  MoveL 728 to (114.51, 182.41, 0) mm, rotated rx 180 ry 0 rz -39.83 deg; joints [46.226, -66.396, 72.244, -0.865, 84.126, 46.311]
  MoveL 729 to (113.63, 182.75, 0) mm, rotated rx 180 ry 0 rz -39.83 deg; joints [46.185, -66.362, 72.194, -0.865, 84.141, 46.27]
  MoveL 730 to (112.75, 183.07, 0) mm, rotated rx 180 ry 0 rz -39.83 deg; joints [46.144, -66.329, 72.147, -0.865, 84.155, 46.229]
  MoveL 731 to (111.7, 183.43, 0) mm, rotated rx -180 ry 0 rz -39.83 deg; joints [46.095, -66.292, 72.093, -0.865, 84.171, 46.18]
  MoveL 732 to (110.64, 183.76, 0) mm, rotated rx 180 ry 0 rz -39.83 deg; joints [46.046, -66.257, 72.043, -0.865, 84.186, 46.13]
  MoveL 733 to (109.56, 184.05, 0) mm, rotated rx 180 ry 0 rz -39.83 deg; joints [45.995, -66.226, 71.997, -0.865, 84.199, 46.079]
  MoveL 734 to (108.47, 184.29, 0) mm, rotated rx 180 ry 0 rz -39.83 deg; joints [45.944, -66.198, 71.957, -0.864, 84.211, 46.028]
  MoveL 735 to (107.39, 184.47, 0) mm, rotated rx 180 ry 0 rz -39.83 deg; joints [45.893, -66.176, 71.924, -0.864, 84.221, 45.977]
  MoveL 736 to (106.3, 184.61, 0) mm, rotated rx 180 ry 0 rz -39.83 deg; joints [45.842, -66.158, 71.897, -0.864, 84.229, 45.925]
  MoveL 737 to (105.21, 184.7, 0) mm, rotated rx 180 ry 0 rz -39.83 deg; joints [45.79, -66.143, 71.874, -0.864, 84.236, 45.874]
  MoveL 738 to (104.14, 184.76, 0) mm, rotated rx 180 ry 0 rz -39.83 deg; joints [45.739, -66.13, 71.855, -0.864, 84.242, 45.822]
  MoveL 739 to (103.53, 184.79, 0) mm, rotated rx 180 ry 0 rz -39.83 deg; joints [45.71, -66.124, 71.846, -0.864, 84.245, 45.794]
  MoveL 740 to (102.92, 184.8, 0) mm, rotated rx 180 ry 0 rz -39.83 deg; joints [45.682, -66.119, 71.838, -0.864, 84.247, 45.765]
  MoveL 741 to (102.31, 184.8, 0) mm, rotated rx -180 ry 0 rz -39.83 deg; joints [45.652, -66.115, 71.832, -0.864, 84.249, 45.736]
  MoveL 742 to (101.69, 184.78, 0) mm, rotated rx -180 ry 0 rz -39.83 deg; joints [45.623, -66.113, 71.828, -0.864, 84.251, 45.706]
  MoveL 743 to (101.69, 184.78, 0) mm, rotated rx -180 ry 0 rz -39.83 deg; joints [45.623, -66.113, 71.828, -0.864, 84.251, 45.706]
  MoveL 744 to (101.07, 184.8, 0) mm, rotated rx 180 ry 0 rz -39.83 deg; joints [45.593, -66.107, 71.818, -0.864, 84.254, 45.676]
  MoveL 745 to (100.46, 184.8, 0) mm, rotated rx 180 ry 0 rz -39.83 deg; joints [45.564, -66.103, 71.811, -0.864, 84.256, 45.647]
  MoveL 746 to (99.86, 184.79, 0) mm, rotated rx -180 ry 0 rz -39.83 deg; joints [45.535, -66.1, 71.807, -0.864, 84.257, 45.618]
  MoveL 747 to (99.25, 184.76, 0) mm, rotated rx 180 ry 0 rz -39.83 deg; joints [45.506, -66.098, 71.803, -0.864, 84.258, 45.589]
  MoveL 748 to (98.18, 184.7, 0) mm, rotated rx 180 ry 0 rz -39.83 deg; joints [45.455, -66.096, 71.799, -0.864, 84.26, 45.538]
  MoveL 749 to (97.09, 184.61, 0) mm, rotated rx 180 ry 0 rz -39.83 deg; joints [45.403, -66.096, 71.798, -0.864, 84.26, 45.486]
  MoveL 750 to (96, 184.47, 0) mm, rotated rx -180 ry 0 rz -39.83 deg; joints [45.35, -66.1, 71.802, -0.864, 84.259, 45.433]
  MoveL 751 to (94.92, 184.29, 0) mm, rotated rx -180 ry 0 rz -39.83 deg; joints [45.298, -66.108, 71.812, -0.864, 84.257, 45.381]
  MoveL 752 to (93.83, 184.05, 0) mm, rotated rx 180 ry 0 rz -39.83 deg; joints [45.245, -66.121, 71.829, -0.864, 84.252, 45.328]
  MoveL 753 to (92.75, 183.76, 0) mm, rotated rx -180 ry 0 rz -39.83 deg; joints [45.193, -66.138, 71.852, -0.864, 84.245, 45.276]
  MoveL 754 to (91.69, 183.43, 0) mm, rotated rx -180 ry 0 rz -39.83 deg; joints [45.141, -66.159, 71.879, -0.864, 84.237, 45.224]
  MoveL 755 to (90.64, 183.07, 0) mm, rotated rx 180 ry 0 rz -39.83 deg; joints [45.089, -66.182, 71.911, -0.864, 84.229, 45.172]
  MoveL 756 to (89.75, 182.75, 0) mm, rotated rx 180 ry 0 rz -39.83 deg; joints [45.046, -66.203, 71.939, -0.864, 84.22, 45.129]
  MoveL 757 to (88.88, 182.41, 0) mm, rotated rx 180 ry 0 rz -39.83 deg; joints [45.003, -66.226, 71.97, -0.864, 84.211, 45.086]
  MoveL 758 to (88.02, 182.04, 0) mm, rotated rx -180 ry 0 rz -39.83 deg; joints [44.96, -66.251, 72.004, -0.864, 84.202, 45.044]
  MoveL 759 to (87.16, 181.64, 0) mm, rotated rx 180 ry 0 rz -39.83 deg; joints [44.917, -66.278, 72.042, -0.864, 84.191, 45.001]
  MoveL 760 to (86.31, 181.19, 0) mm, rotated rx 180 ry 0 rz -39.83 deg; joints [44.875, -66.31, 72.086, -0.864, 84.178, 44.959]
  MoveL 761 to (85.46, 180.71, 0) mm, rotated rx 180 ry 0 rz -39.83 deg; joints [44.832, -66.345, 72.134, -0.864, 84.164, 44.916]
  MoveL 762 to (84.63, 180.2, 0) mm, rotated rx 180 ry 0 rz -39.83 deg; joints [44.79, -66.382, 72.185, -0.864, 84.149, 44.875]
  MoveL 763 to (83.81, 179.68, 0) mm, rotated rx 180 ry 0 rz -39.83 deg; joints [44.749, -66.421, 72.239, -0.864, 84.134, 44.833]
  MoveL 764 to (83.1, 179.21, 0) mm, rotated rx 180 ry 0 rz -39.83 deg; joints [44.713, -66.455, 72.287, -0.864, 84.12, 44.798]
  MoveL 765 to (82.4, 178.72, 0) mm, rotated rx -180 ry 0 rz -39.83 deg; joints [44.677, -66.491, 72.336, -0.864, 84.106, 44.762]
  MoveL 766 to (81.72, 178.23, 0) mm, rotated rx 180 ry 0 rz -39.83 deg; joints [44.642, -66.528, 72.388, -0.864, 84.091, 44.727]
  MoveL 767 to (81.05, 177.71, 0) mm, rotated rx -180 ry 0 rz -39.83 deg; joints [44.608, -66.567, 72.441, -0.864, 84.076, 44.693]
  MoveL 768 to (80.23, 177.02, 0) mm, rotated rx 180 ry 0 rz -39.83 deg; joints [44.566, -66.619, 72.514, -0.864, 84.055, 44.651]
  MoveL 769 to (79.45, 176.29, 0) mm, rotated rx 180 ry 0 rz -39.83 deg; joints [44.525, -66.675, 72.591, -0.864, 84.033, 44.611]
  MoveL 770 to (78.71, 175.53, 0) mm, rotated rx -180 ry 0 rz -39.83 deg; joints [44.486, -66.734, 72.673, -0.864, 84.009, 44.572]
  MoveL 771 to (78.02, 174.73, 0) mm, rotated rx 180 ry 0 rz -39.83 deg; joints [44.449, -66.797, 72.76, -0.864, 83.984, 44.536]
  MoveL 772 to (77.69, 174.31, 0) mm, rotated rx 180 ry 0 rz -39.83 deg; joints [44.431, -66.83, 72.806, -0.864, 83.971, 44.518]
  MoveL 773 to (77.38, 173.88, 0) mm, rotated rx -180 ry 0 rz -39.83 deg; joints [44.414, -66.864, 72.854, -0.864, 83.957, 44.501]
  MoveL 774 to (77.09, 173.42, 0) mm, rotated rx 180 ry 0 rz -39.83 deg; joints [44.398, -66.901, 72.905, -0.864, 83.943, 44.485]
  MoveL 775 to (76.83, 172.93, 0) mm, rotated rx -180 ry 0 rz -39.83 deg; joints [44.383, -66.94, 72.96, -0.864, 83.927, 44.471]
  MoveL 776 to (76.65, 172.52, 0) mm, rotated rx 180 ry 0 rz -39.83 deg; joints [44.373, -66.974, 73.007, -0.864, 83.913, 44.46]
  MoveL 777 to (76.49, 172.09, 0) mm, rotated rx -180 ry 0 rz -39.83 deg; joints [44.363, -67.009, 73.056, -0.864, 83.899, 44.451]
  MoveL 778 to (76.36, 171.66, 0) mm, rotated rx 180 ry 0 rz -39.83 deg; joints [44.355, -67.045, 73.106, -0.864, 83.885, 44.443]
  MoveL 779 to (76.26, 171.24, 0) mm, rotated rx -180 ry 0 rz -39.83 deg; joints [44.348, -67.08, 73.155, -0.864, 83.871, 44.436]
  MoveL 780 to (76.2, 170.92, 0) mm, rotated rx 180 ry 0 rz -39.83 deg; joints [44.343, -67.107, 73.192, -0.864, 83.861, 44.432]
  MoveL 781 to (76.15, 170.61, 0) mm, rotated rx -180 ry 0 rz -39.83 deg; joints [44.339, -67.133, 73.229, -0.864, 83.85, 44.428]
  MoveL 782 to (76.11, 170.29, 0) mm, rotated rx 180 ry 0 rz -39.83 deg; joints [44.336, -67.16, 73.266, -0.864, 83.84, 44.425]
  MoveL 783 to (76.08, 169.97, 0) mm, rotated rx 180 ry 0 rz -39.83 deg; joints [44.333, -67.187, 73.304, -0.864, 83.829, 44.422]
  MoveL 784 to (76.06, 169.58, 0) mm, rotated rx 180 ry 0 rz -39.83 deg; joints [44.33, -67.22, 73.35, -0.864, 83.816, 44.419]
  MoveL 785 to (76.05, 169.18, 0) mm, rotated rx 180 ry 0 rz -39.83 deg; joints [44.327, -67.254, 73.397, -0.864, 83.802, 44.417]
  MoveL 786 to (76.05, 168.78, 0) mm, rotated rx 180 ry 0 rz -39.83 deg; joints [44.325, -67.288, 73.445, -0.864, 83.788, 44.415]
  MoveL 787 to (76.07, 168.37, 0) mm, rotated rx 180 ry 0 rz -39.83 deg; joints [44.324, -67.323, 73.494, -0.864, 83.775, 44.414]
  MoveL 788 to (76.11, 167.98, 0) mm, rotated rx -180 ry 0 rz -39.83 deg; joints [44.324, -67.356, 73.541, -0.864, 83.761, 44.415]
  MoveL 789 to (76.17, 167.59, 0) mm, rotated rx 180 ry 0 rz -39.83 deg; joints [44.325, -67.39, 73.588, -0.864, 83.748, 44.416]
  MoveL 790 to (76.26, 167.21, 0) mm, rotated rx -180 ry 0 rz -39.83 deg; joints [44.328, -67.423, 73.634, -0.864, 83.735, 44.418]
  MoveL 791 to (76.37, 166.84, 0) mm, rotated rx 180 ry 0 rz -39.83 deg; joints [44.331, -67.456, 73.679, -0.864, 83.722, 44.422]
  MoveL 792 to (76.54, 166.39, 0) mm, rotated rx -180 ry 0 rz -39.83 deg; joints [44.337, -67.495, 73.734, -0.864, 83.707, 44.428]
  MoveL 793 to (76.74, 165.96, 0) mm, rotated rx -180 ry 0 rz -39.83 deg; joints [44.345, -67.534, 73.789, -0.864, 83.691, 44.436]
  MoveL 794 to (76.97, 165.53, 0) mm, rotated rx -180 ry 0 rz -39.83 deg; joints [44.354, -67.572, 73.842, -0.864, 83.676, 44.445]
  MoveL 795 to (77.22, 165.11, 0) mm, rotated rx 180 ry 0 rz -39.83 deg; joints [44.364, -67.61, 73.895, -0.864, 83.661, 44.456]
  MoveL 796 to (77.53, 164.64, 0) mm, rotated rx -180 ry 0 rz -39.83 deg; joints [44.376, -67.653, 73.955, -0.864, 83.644, 44.468]
  MoveL 797 to (77.86, 164.18, 0) mm, rotated rx 180 ry 0 rz -39.83 deg; joints [44.39, -67.694, 74.014, -0.864, 83.628, 44.482]
  MoveL 798 to (78.2, 163.73, 0) mm, rotated rx -180 ry 0 rz -39.83 deg; joints [44.404, -67.735, 74.071, -0.864, 83.612, 44.497]
  MoveL 799 to (78.57, 163.3, 0) mm, rotated rx 180 ry 0 rz -39.83 deg; joints [44.42, -67.774, 74.126, -0.864, 83.596, 44.513]
  MoveL 800 to (79, 162.85, 0) mm, rotated rx -180 ry 0 rz -39.83 deg; joints [44.439, -67.817, 74.185, -0.864, 83.579, 44.532]
  MoveL 801 to (79.47, 162.42, 0) mm, rotated rx 180 ry 0 rz -39.83 deg; joints [44.459, -67.857, 74.241, -0.864, 83.563, 44.552]
  MoveL 802 to (79.95, 162.01, 0) mm, rotated rx 180 ry 0 rz -39.83 deg; joints [44.48, -67.896, 74.296, -0.865, 83.548, 44.574]
  MoveL 803 to (80.45, 161.62, 0) mm, rotated rx 180 ry 0 rz -39.83 deg; joints [44.503, -67.933, 74.348, -0.865, 83.534, 44.596]
  MoveL 804 to (81.09, 161.15, 0) mm, rotated rx 180 ry 0 rz -39.83 deg; joints [44.532, -67.978, 74.411, -0.865, 83.516, 44.626]
  MoveL 805 to (81.75, 160.71, 0) mm, rotated rx 180 ry 0 rz -39.83 deg; joints [44.562, -68.02, 74.471, -0.865, 83.499, 44.656]
  MoveL 806 to (82.43, 160.29, 0) mm, rotated rx 180 ry 0 rz -39.83 deg; joints [44.593, -68.061, 74.528, -0.865, 83.483, 44.687]
  MoveL 807 to (83.12, 159.89, 0) mm, rotated rx 180 ry 0 rz -39.83 deg; joints [44.624, -68.101, 74.584, -0.865, 83.467, 44.719]
  MoveL 808 to (83.7, 159.57, 0) mm, rotated rx 180 ry 0 rz -39.83 deg; joints [44.651, -68.133, 74.629, -0.865, 83.455, 44.746]
  MoveL 809 to (84.29, 159.25, 0) mm, rotated rx 180 ry 0 rz -39.83 deg; joints [44.678, -68.165, 74.673, -0.865, 83.442, 44.773]
  MoveL 810 to (84.89, 158.95, 0) mm, rotated rx 180 ry 0 rz -39.83 deg; joints [44.705, -68.195, 74.716, -0.865, 83.43, 44.801]
  MoveL 811 to (85.49, 158.67, 0) mm, rotated rx 180 ry 0 rz -39.83 deg; joints [44.734, -68.224, 74.757, -0.865, 83.419, 44.829]
  MoveL 812 to (86.31, 158.32, 0) mm, rotated rx 180 ry 0 rz -39.83 deg; joints [44.772, -68.26, 74.807, -0.865, 83.405, 44.868]
  MoveL 813 to (87.14, 157.99, 0) mm, rotated rx 180 ry 0 rz -39.83 deg; joints [44.811, -68.293, 74.855, -0.865, 83.392, 44.907]
  MoveL 814 to (87.99, 157.69, 0) mm, rotated rx 180 ry 0 rz -39.83 deg; joints [44.85, -68.325, 74.9, -0.865, 83.379, 44.946]
  MoveL 815 to (88.83, 157.41, 0) mm, rotated rx 180 ry 0 rz -39.83 deg; joints [44.89, -68.356, 74.943, -0.865, 83.367, 44.987]
  MoveL 816 to (89.62, 157.16, 0) mm, rotated rx -180 ry 0 rz -39.83 deg; joints [44.927, -68.383, 74.981, -0.865, 83.356, 45.024]
  MoveL 817 to (90.4, 156.92, 0) mm, rotated rx 180 ry 0 rz -39.83 deg; joints [44.964, -68.409, 75.018, -0.865, 83.346, 45.061]
  MoveL 818 to (91.19, 156.7, 0) mm, rotated rx 180 ry 0 rz -39.83 deg; joints [45.002, -68.434, 75.053, -0.865, 83.336, 45.099]
  MoveL 819 to (91.99, 156.5, 0) mm, rotated rx 180 ry 0 rz -39.83 deg; joints [45.04, -68.457, 75.086, -0.865, 83.327, 45.137]
  MoveL 820 to (92.82, 156.31, 0) mm, rotated rx 180 ry 0 rz -39.83 deg; joints [45.08, -68.479, 75.118, -0.865, 83.318, 45.177]
  MoveL 821 to (93.66, 156.14, 0) mm, rotated rx 180 ry 0 rz -39.83 deg; joints [45.12, -68.499, 75.147, -0.865, 83.31, 45.217]
  MoveL 822 to (94.51, 155.99, 0) mm, rotated rx 180 ry 0 rz -39.83 deg; joints [45.16, -68.518, 75.174, -0.865, 83.302, 45.258]
  MoveL 823 to (95.35, 155.86, 0) mm, rotated rx 180 ry 0 rz -39.83 deg; joints [45.201, -68.535, 75.199, -0.866, 83.295, 45.298]
  MoveL 824 to (96.38, 155.71, 0) mm, rotated rx 180 ry 0 rz -39.83 deg; joints [45.25, -68.555, 75.227, -0.866, 83.288, 45.348]
  MoveL 825 to (97.41, 155.59, 0) mm, rotated rx 180 ry 0 rz -39.83 deg; joints [45.3, -68.572, 75.252, -0.866, 83.28, 45.398]
  MoveL 826 to (98.44, 155.49, 0) mm, rotated rx -180 ry 0 rz -39.83 deg; joints [45.35, -68.588, 75.275, -0.866, 83.274, 45.448]
  MoveL 827 to (99.47, 155.42, 0) mm, rotated rx 180 ry 0 rz -39.83 deg; joints [45.4, -68.601, 75.294, -0.866, 83.269, 45.498]
  MoveL 828 to (100.02, 155.4, 0) mm, rotated rx 180 ry 0 rz -39.83 deg; joints [45.427, -68.606, 75.303, -0.866, 83.266, 45.525]
  MoveL 829 to (100.58, 155.38, 0) mm, rotated rx 180 ry 0 rz -39.83 deg; joints [45.454, -68.612, 75.311, -0.866, 83.264, 45.552]
  MoveL 830 to (101.14, 155.37, 0) mm, rotated rx -180 ry 0 rz -39.83 deg; joints [45.481, -68.616, 75.318, -0.866, 83.262, 45.579]
  MoveL 831 to (101.69, 155.36, 0) mm, rotated rx 180 ry 0 rz -39.83 deg; joints [45.508, -68.621, 75.325, -0.866, 83.26, 45.607]
  Establecer velocidad (1000.0 mm/s)
  MoveL 832 to (101.69, 155.36, 0) mm, rotated rx 180 ry 0 rz -39.83 deg; joints [45.508, -68.621, 75.325, -0.866, 83.26, 45.607]
  MoveL 833 to (101.69, 155.36, 20) mm, rotated rx 180 ry 0 rz -39.83 deg; joints [45.523, -68.888, 73.963, -0.863, 84.889, 45.597]

--- program P_in_2 (robot KUKA KR 16 2) ---
  Suave(1)
  Establecer velocidad (1000.0 mm/s)
  Est. Ref.: Frame 2
  Est. herr: Plumon_ensamble
  Mostrar Plumon_ensamble
  MoveJ 1 to (138.11, 152.35, 20) mm, rotated rx -180 ry 0 rz -39.83 deg; joints [47.298, -69.343, 74.631, -0.864, 84.703, 47.375]
  MoveL 2 to (138.11, 152.35, 20) mm, rotated rx -180 ry 0 rz -39.83 deg; joints [47.298, -69.343, 74.631, -0.864, 84.703, 47.375]
  MoveL 3 to (138.11, 152.35, 0) mm, rotated rx 180 ry 0 rz -39.83 deg; joints [47.283, -69.071, 75.989, -0.867, 83.072, 47.385]
  MoveL 4 to (138.11, 152.35, 0) mm, rotated rx 180 ry 0 rz -39.83 deg; joints [47.283, -69.071, 75.989, -0.867, 83.072, 47.385]
  Establecer velocidad (50.0 mm/s)
  MoveL 5 to (138.89, 152.07, 0) mm, rotated rx -180 ry 0 rz -39.83 deg; joints [47.321, -69.098, 76.027, -0.867, 83.062, 47.422]
  MoveL 6 to (139.65, 151.76, 0) mm, rotated rx -180 ry 0 rz -39.83 deg; joints [47.358, -69.127, 76.067, -0.867, 83.051, 47.459]
  MoveL 7 to (140.41, 151.43, 0) mm, rotated rx 180 ry 0 rz -39.83 deg; joints [47.394, -69.157, 76.11, -0.867, 83.039, 47.496]
  MoveL 8 to (141.16, 151.09, 0) mm, rotated rx 180 ry 0 rz -39.83 deg; joints [47.43, -69.189, 76.155, -0.867, 83.027, 47.532]
  MoveL 9 to (142.11, 150.62, 0) mm, rotated rx 180 ry 0 rz -39.83 deg; joints [47.476, -69.232, 76.215, -0.867, 83.011, 47.578]
  MoveL 10 to (143.04, 150.14, 0) mm, rotated rx 180 ry 0 rz -39.83 deg; joints [47.521, -69.277, 76.276, -0.867, 82.994, 47.623]
  MoveL 11 to (143.96, 149.63, 0) mm, rotated rx -180 ry 0 rz -39.83 deg; joints [47.565, -69.323, 76.341, -0.867, 82.977, 47.668]
  MoveL 12 to (144.87, 149.1, 0) mm, rotated rx 180 ry 0 rz -39.83 deg; joints [47.609, -69.37, 76.407, -0.867, 82.959, 47.712]
  MoveL 13 to (146, 148.42, 0) mm, rotated rx 180 ry 0 rz -39.83 deg; joints [47.663, -69.432, 76.492, -0.867, 82.936, 47.766]
  MoveL 14 to (147.1, 147.68, 0) mm, rotated rx 180 ry 0 rz -39.83 deg; joints [47.716, -69.498, 76.583, -0.867, 82.912, 47.819]
  MoveL 15 to (148.15, 146.89, 0) mm, rotated rx 180 ry 0 rz -39.83 deg; joints [47.766, -69.568, 76.68, -0.867, 82.886, 47.87]
  MoveL 16 to (149.12, 146.01, 0) mm, rotated rx 180 ry 0 rz -39.83 deg; joints [47.812, -69.645, 76.786, -0.867, 82.858, 47.916]
  MoveL 17 to (149.82, 145.25, 0) mm, rotated rx 180 ry 0 rz -39.83 deg; joints [47.845, -69.712, 76.877, -0.867, 82.834, 47.95]
  MoveL 18 to (150.48, 144.46, 0) mm, rotated rx 180 ry 0 rz -39.83 deg; joints [47.876, -69.781, 76.972, -0.867, 82.809, 47.982]
  MoveL 19 to (151.13, 143.64, 0) mm, rotated rx 180 ry 0 rz -39.83 deg; joints [47.907, -69.852, 77.069, -0.868, 82.783, 48.013]
  MoveL 20 to (151.78, 142.82, 0) mm, rotated rx -180 ry 0 rz -39.83 deg; joints [47.937, -69.923, 77.165, -0.868, 82.758, 48.043]
  MoveL 21 to (152.63, 141.8, 0) mm, rotated rx -180 ry 0 rz -39.83 deg; joints [47.978, -70.011, 77.286, -0.868, 82.726, 48.084]
  MoveL 22 to (153.49, 140.78, 0) mm, rotated rx -180 ry 0 rz -39.83 deg; joints [48.019, -70.099, 77.405, -0.868, 82.695, 48.126]
  MoveL 23 to (154.33, 139.76, 0) mm, rotated rx 180 ry 0 rz -39.83 deg; joints [48.058, -70.187, 77.526, -0.868, 82.663, 48.166]
  MoveL 24 to (155.11, 138.69, 0) mm, rotated rx 180 ry 0 rz -39.83 deg; joints [48.095, -70.279, 77.651, -0.868, 82.631, 48.203]
  MoveL 25 to (155.71, 137.74, 0) mm, rotated rx 180 ry 0 rz -39.83 deg; joints [48.123, -70.361, 77.761, -0.868, 82.602, 48.232]
  MoveL 26 to (156.26, 136.75, 0) mm, rotated rx 180 ry 0 rz -39.83 deg; joints [48.149, -70.445, 77.876, -0.868, 82.573, 48.258]
  MoveL 27 to (156.76, 135.74, 0) mm, rotated rx -180 ry 0 rz -39.83 deg; joints [48.172, -70.532, 77.993, -0.868, 82.543, 48.282]
  MoveL 28 to (157.24, 134.7, 0) mm, rotated rx 180 ry 0 rz -39.83 deg; joints [48.194, -70.62, 78.111, -0.868, 82.512, 48.304]
  MoveL 29 to (157.83, 133.33, 0) mm, rotated rx -180 ry 0 rz -39.83 deg; joints [48.222, -70.736, 78.268, -0.868, 82.472, 48.332]
  MoveL 30 to (158.37, 131.95, 0) mm, rotated rx 180 ry 0 rz -39.83 deg; joints [48.246, -70.853, 78.426, -0.868, 82.432, 48.358]
  MoveL 31 to (158.85, 130.54, 0) mm, rotated rx 180 ry 0 rz -39.83 deg; joints [48.268, -70.972, 78.586, -0.868, 82.392, 48.38]
  MoveL 32 to (159.24, 129.11, 0) mm, rotated rx 180 ry 0 rz -39.83 deg; joints [48.285, -71.093, 78.747, -0.868, 82.351, 48.397]
  MoveL 33 to (159.49, 127.9, 0) mm, rotated rx 180 ry 0 rz -39.83 deg; joints [48.296, -71.195, 78.883, -0.868, 82.317, 48.408]
  MoveL 34 to (159.67, 126.67, 0) mm, rotated rx 180 ry 0 rz -39.83 deg; joints [48.303, -71.298, 79.021, -0.868, 82.283, 48.416]
  MoveL 35 to (159.81, 125.43, 0) mm, rotated rx 180 ry 0 rz -39.83 deg; joints [48.308, -71.402, 79.159, -0.869, 82.249, 48.422]
  MoveL 36 to (159.9, 124.19, 0) mm, rotated rx -180 ry 0 rz -39.83 deg; joints [48.31, -71.506, 79.297, -0.869, 82.215, 48.425]
  MoveL 37 to (159.96, 123.02, 0) mm, rotated rx -180 ry 0 rz -39.83 deg; joints [48.311, -71.603, 79.426, -0.869, 82.183, 48.426]
  MoveL 38 to (159.99, 121.86, 0) mm, rotated rx 180 ry 0 rz -39.83 deg; joints [48.311, -71.701, 79.555, -0.869, 82.151, 48.426]
  MoveL 39 to (159.97, 120.69, 0) mm, rotated rx 180 ry 0 rz -39.83 deg; joints [48.308, -71.798, 79.684, -0.869, 82.12, 48.424]
  MoveL 40 to (159.9, 119.53, 0) mm, rotated rx 180 ry 0 rz -39.83 deg; joints [48.303, -71.894, 79.811, -0.869, 82.089, 48.419]
  MoveL 41 to (159.71, 117.85, 0) mm, rotated rx -180 ry 0 rz -39.83 deg; joints [48.29, -72.034, 79.995, -0.869, 82.044, 48.407]
  MoveL 42 to (159.41, 116.18, 0) mm, rotated rx 180 ry 0 rz -39.83 deg; joints [48.272, -72.172, 80.177, -0.869, 82.001, 48.39]
  MoveL 43 to (159.03, 114.52, 0) mm, rotated rx 180 ry 0 rz -39.83 deg; joints [48.25, -72.309, 80.357, -0.869, 81.958, 48.368]
  MoveL 44 to (158.57, 112.88, 0) mm, rotated rx -180 ry 0 rz -39.83 deg; joints [48.224, -72.445, 80.534, -0.869, 81.916, 48.343]
  MoveL 45 to (158.12, 111.47, 0) mm, rotated rx 180 ry 0 rz -39.83 deg; joints [48.198, -72.561, 80.686, -0.869, 81.88, 48.318]
  MoveL 46 to (157.6, 110.08, 0) mm, rotated rx 180 ry 0 rz -39.83 deg; joints [48.169, -72.676, 80.835, -0.869, 81.845, 48.29]
  MoveL 47 to (157, 108.73, 0) mm, rotated rx -180 ry 0 rz -39.83 deg; joints [48.136, -72.786, 80.978, -0.869, 81.811, 48.257]
  MoveL 48 to (156.31, 107.43, 0) mm, rotated rx 180 ry 0 rz -39.83 deg; joints [48.098, -72.892, 81.116, -0.87, 81.779, 48.219]
  MoveL 49 to (155.34, 105.97, 0) mm, rotated rx -180 ry 0 rz -39.83 deg; joints [48.046, -73.01, 81.268, -0.87, 81.744, 48.168]
  MoveL 50 to (154.22, 104.62, 0) mm, rotated rx 180 ry 0 rz -39.83 deg; joints [47.986, -73.119, 81.408, -0.87, 81.712, 48.108]
  MoveL 51 to (152.99, 103.37, 0) mm, rotated rx 180 ry 0 rz -39.83 deg; joints [47.92, -73.219, 81.536, -0.87, 81.683, 48.043]
  MoveL 52 to (151.65, 102.24, 0) mm, rotated rx 180 ry 0 rz -39.83 deg; joints [47.849, -73.309, 81.651, -0.87, 81.657, 47.972]
  MoveL 53 to (150.39, 101.33, 0) mm, rotated rx 180 ry 0 rz -39.83 deg; joints [47.783, -73.38, 81.742, -0.87, 81.636, 47.906]
  MoveL 54 to (149.08, 100.52, 0) mm, rotated rx 180 ry 0 rz -39.83 deg; joints [47.713, -73.443, 81.821, -0.87, 81.619, 47.837]
  MoveL 55 to (147.72, 99.8, 0) mm, rotated rx -180 ry 0 rz -39.83 deg; joints [47.642, -73.498, 81.891, -0.87, 81.603, 47.765]
  MoveL 56 to (146.32, 99.18, 0) mm, rotated rx 180 ry 0 rz -39.83 deg; joints [47.568, -73.545, 81.95, -0.87, 81.59, 47.692]
  MoveL 57 to (145.08, 98.71, 0) mm, rotated rx 180 ry 0 rz -39.83 deg; joints [47.503, -73.579, 81.992, -0.87, 81.581, 47.627]
  MoveL 58 to (143.83, 98.32, 0) mm, rotated rx 180 ry 0 rz -39.83 deg; joints [47.437, -73.607, 82.027, -0.87, 81.573, 47.562]
  MoveL 59 to (142.55, 97.98, 0) mm, rotated rx 180 ry 0 rz -39.83 deg; joints [47.371, -73.63, 82.055, -0.87, 81.567, 47.495]
  MoveL 60 to (141.26, 97.71, 0) mm, rotated rx 180 ry 0 rz -39.83 deg; joints [47.303, -73.647, 82.075, -0.87, 81.563, 47.428]
  MoveL 61 to (139.77, 97.48, 0) mm, rotated rx -180 ry 0 rz -39.83 deg; joints [47.226, -73.661, 82.091, -0.87, 81.56, 47.35]
  MoveL 62 to (138.27, 97.33, 0) mm, rotated rx 180 ry 0 rz -39.83 deg; joints [47.148, -73.667, 82.097, -0.87, 81.559, 47.273]
  MoveL 63 to (136.77, 97.27, 0) mm, rotated rx 180 ry 0 rz -39.83 deg; joints [47.07, -73.666, 82.093, -0.87, 81.56, 47.195]
  MoveL 64 to (135.27, 97.31, 0) mm, rotated rx 180 ry 0 rz -39.83 deg; joints [46.993, -73.656, 82.078, -0.87, 81.564, 47.117]
  MoveL 65 to (133.81, 97.45, 0) mm, rotated rx 180 ry 0 rz -39.83 deg; joints [46.919, -73.638, 82.054, -0.87, 81.57, 47.043]
  MoveL 66 to (132.37, 97.68, 0) mm, rotated rx 180 ry 0 rz -39.83 deg; joints [46.845, -73.613, 82.019, -0.87, 81.578, 46.969]
  MoveL 67 to (130.95, 97.99, 0) mm, rotated rx 180 ry 0 rz -39.83 deg; joints [46.773, -73.58, 81.975, -0.87, 81.588, 46.896]
  MoveL 68 to (129.54, 98.38, 0) mm, rotated rx 180 ry 0 rz -39.83 deg; joints [46.701, -73.542, 81.923, -0.87, 81.6, 46.825]
  MoveL 69 to (128.37, 98.76, 0) mm, rotated rx 180 ry 0 rz -39.83 deg; joints [46.642, -73.504, 81.874, -0.87, 81.612, 46.766]
  MoveL 70 to (127.22, 99.19, 0) mm, rotated rx -180 ry 0 rz -39.83 deg; joints [46.584, -73.463, 81.818, -0.87, 81.624, 46.708]
  MoveL 71 to (126.1, 99.69, 0) mm, rotated rx 180 ry 0 rz -39.83 deg; joints [46.528, -73.416, 81.757, -0.87, 81.639, 46.651]
  MoveL 72 to (125.01, 100.24, 0) mm, rotated rx -180 ry 0 rz -39.83 deg; joints [46.474, -73.365, 81.689, -0.87, 81.654, 46.597]
  MoveL 73 to (123.6, 101.09, 0) mm, rotated rx 180 ry 0 rz -39.83 deg; joints [46.405, -73.288, 81.587, -0.869, 81.678, 46.527]
  MoveL 74 to (122.25, 102.03, 0) mm, rotated rx 180 ry 0 rz -39.83 deg; joints [46.339, -73.203, 81.475, -0.869, 81.704, 46.461]
  MoveL 75 to (120.95, 103.04, 0) mm, rotated rx 180 ry 0 rz -39.83 deg; joints [46.275, -73.112, 81.355, -0.869, 81.732, 46.397]
  MoveL 76 to (119.68, 104.1, 0) mm, rotated rx 180 ry 0 rz -39.83 deg; joints [46.214, -73.017, 81.23, -0.869, 81.761, 46.335]
  MoveL 77 to (118.34, 105.29, 0) mm, rotated rx -180 ry 0 rz -39.83 deg; joints [46.15, -72.911, 81.09, -0.869, 81.794, 46.27]
  MoveL 78 to (117.04, 106.52, 0) mm, rotated rx -180 ry 0 rz -39.83 deg; joints [46.088, -72.801, 80.946, -0.869, 81.828, 46.208]
  MoveL 79 to (115.79, 107.81, 0) mm, rotated rx 180 ry 0 rz -39.83 deg; joints [46.029, -72.688, 80.796, -0.869, 81.864, 46.148]
  MoveL 80 to (114.62, 109.16, 0) mm, rotated rx 180 ry 0 rz -39.83 deg; joints [45.974, -72.569, 80.639, -0.869, 81.901, 46.093]
  MoveL 81 to (113.74, 110.29, 0) mm, rotated rx 180 ry 0 rz -39.83 deg; joints [45.934, -72.469, 80.507, -0.869, 81.932, 46.052]
  MoveL 82 to (112.92, 111.47, 0) mm, rotated rx -180 ry 0 rz -39.83 deg; joints [45.896, -72.366, 80.371, -0.869, 81.965, 46.014]
  MoveL 83 to (112.15, 112.69, 0) mm, rotated rx 180 ry 0 rz -39.83 deg; joints [45.862, -72.26, 80.231, -0.869, 81.999, 45.979]
  MoveL 84 to (111.43, 113.95, 0) mm, rotated rx -180 ry 0 rz -39.83 deg; joints [45.83, -72.152, 80.088, -0.868, 82.033, 45.947]
  MoveL 85 to (110.6, 115.55, 0) mm, rotated rx 180 ry 0 rz -39.83 deg; joints [45.794, -72.013, 79.904, -0.868, 82.078, 45.911]
  MoveL 86 to (109.85, 117.2, 0) mm, rotated rx 180 ry 0 rz -39.83 deg; joints [45.763, -71.872, 79.716, -0.868, 82.123, 45.879]
  MoveL 87 to (109.19, 118.88, 0) mm, rotated rx 180 ry 0 rz -39.83 deg; joints [45.736, -71.728, 79.525, -0.868, 82.17, 45.851]
  MoveL 88 to (108.63, 120.6, 0) mm, rotated rx 180 ry 0 rz -39.83 deg; joints [45.715, -71.581, 79.33, -0.868, 82.218, 45.829]
  MoveL 89 to (108.12, 122.52, 0) mm, rotated rx 180 ry 0 rz -39.83 deg; joints [45.697, -71.418, 79.112, -0.868, 82.272, 45.81]
  MoveL 90 to (107.73, 124.48, 0) mm, rotated rx 180 ry 0 rz -39.83 deg; joints [45.685, -71.252, 78.892, -0.868, 82.327, 45.797]
  MoveL 91 to (107.46, 126.46, 0) mm, rotated rx -180 ry 0 rz -39.83 deg; joints [45.679, -71.086, 78.67, -0.868, 82.382, 45.79]
  MoveL 92 to (107.3, 128.45, 0) mm, rotated rx -180 ry 0 rz -39.83 deg; joints [45.679, -70.918, 78.446, -0.867, 82.439, 45.789]
  MoveL 93 to (107.26, 129.89, 0) mm, rotated rx 180 ry 0 rz -39.83 deg; joints [45.682, -70.798, 78.285, -0.867, 82.479, 45.792]
  MoveL 94 to (107.28, 131.32, 0) mm, rotated rx 180 ry 0 rz -39.83 deg; joints [45.689, -70.678, 78.125, -0.867, 82.52, 45.799]
  MoveL 95 to (107.38, 132.75, 0) mm, rotated rx 180 ry 0 rz -39.83 deg; joints [45.7, -70.559, 77.965, -0.867, 82.561, 45.809]
  MoveL 96 to (107.56, 134.17, 0) mm, rotated rx -180 ry 0 rz -39.83 deg; joints [45.714, -70.442, 77.807, -0.867, 82.601, 45.823]
  MoveL 97 to (107.88, 135.74, 0) mm, rotated rx 180 ry 0 rz -39.83 deg; joints [45.736, -70.312, 77.634, -0.867, 82.646, 45.844]
  MoveL 98 to (108.3, 137.28, 0) mm, rotated rx 180 ry 0 rz -39.83 deg; joints [45.763, -70.185, 77.464, -0.867, 82.689, 45.87]
  MoveL 99 to (108.82, 138.8, 0) mm, rotated rx 180 ry 0 rz -39.83 deg; joints [45.795, -70.061, 77.297, -0.867, 82.733, 45.901]
  MoveL 100 to (109.43, 140.29, 0) mm, rotated rx 180 ry 0 rz -39.83 deg; joints [45.83, -69.94, 77.134, -0.867, 82.775, 45.936]
  MoveL 101 to (110.26, 142.02, 0) mm, rotated rx 180 ry 0 rz -39.83 deg; joints [45.878, -69.8, 76.945, -0.867, 82.824, 45.983]
  MoveL 102 to (111.22, 143.67, 0) mm, rotated rx 180 ry 0 rz -39.83 deg; joints [45.932, -69.667, 76.766, -0.867, 82.871, 46.036]
  MoveL 103 to (112.32, 145.24, 0) mm, rotated rx -180 ry 0 rz -39.83 deg; joints [45.991, -69.542, 76.597, -0.867, 82.915, 46.095]
  MoveL 104 to (113.56, 146.68, 0) mm, rotated rx 180 ry 0 rz -39.83 deg; joints [46.058, -69.428, 76.444, -0.867, 82.956, 46.161]
  MoveL 105 to (114.42, 147.52, 0) mm, rotated rx 180 ry 0 rz -39.83 deg; joints [46.103, -69.362, 76.355, -0.867, 82.979, 46.206]
  MoveL 106 to (115.34, 148.31, 0) mm, rotated rx 180 ry 0 rz -39.83 deg; joints [46.151, -69.301, 76.273, -0.867, 83.001, 46.253]
  MoveL 107 to (116.29, 149.04, 0) mm, rotated rx 180 ry 0 rz -39.83 deg; joints [46.201, -69.244, 76.197, -0.867, 83.021, 46.303]
  MoveL 108 to (117.29, 149.74, 0) mm, rotated rx -180 ry 0 rz -39.83 deg; joints [46.252, -69.191, 76.126, -0.867, 83.04, 46.353]
  MoveL 109 to (118.22, 150.33, 0) mm, rotated rx 180 ry 0 rz -39.83 deg; joints [46.3, -69.146, 76.066, -0.867, 83.056, 46.401]
  MoveL 110 to (119.17, 150.89, 0) mm, rotated rx 180 ry 0 rz -39.83 deg; joints [46.348, -69.104, 76.01, -0.867, 83.071, 46.449]
  MoveL 111 to (120.15, 151.4, 0) mm, rotated rx -180 ry 0 rz -39.83 deg; joints [46.398, -69.066, 75.959, -0.867, 83.084, 46.499]
  MoveL 112 to (121.15, 151.87, 0) mm, rotated rx 180 ry 0 rz -39.83 deg; joints [46.449, -69.033, 75.915, -0.867, 83.096, 46.549]
  MoveL 113 to (122.06, 152.23, 0) mm, rotated rx 180 ry 0 rz -39.83 deg; joints [46.494, -69.006, 75.88, -0.867, 83.105, 46.595]
  MoveL 114 to (122.98, 152.55, 0) mm, rotated rx 180 ry 0 rz -39.83 deg; joints [46.541, -68.984, 75.851, -0.867, 83.113, 46.641]
  MoveL 115 to (123.92, 152.83, 0) mm, rotated rx 180 ry 0 rz -39.83 deg; joints [46.588, -68.965, 75.826, -0.867, 83.119, 46.688]
  MoveL 116 to (124.88, 153.06, 0) mm, rotated rx -180 ry 0 rz -39.83 deg; joints [46.635, -68.951, 75.807, -0.867, 83.124, 46.736]
  MoveL 117 to (125.65, 153.22, 0) mm, rotated rx -180 ry 0 rz -39.83 deg; joints [46.674, -68.941, 75.796, -0.867, 83.127, 46.774]
  MoveL 118 to (126.43, 153.34, 0) mm, rotated rx -180 ry 0 rz -39.83 deg; joints [46.713, -68.935, 75.787, -0.867, 83.129, 46.813]
  MoveL 119 to (127.22, 153.45, 0) mm, rotated rx -180 ry 0 rz -39.83 deg; joints [46.751, -68.93, 75.782, -0.867, 83.13, 46.852]
  MoveL 120 to (128, 153.53, 0) mm, rotated rx 180 ry 0 rz -39.83 deg; joints [46.79, -68.926, 75.778, -0.867, 83.131, 46.89]
  MoveL 121 to (128.52, 153.58, 0) mm, rotated rx 180 ry 0 rz -39.83 deg; joints [46.816, -68.925, 75.777, -0.867, 83.131, 46.916]
  MoveL 122 to (129.05, 153.62, 0) mm, rotated rx 180 ry 0 rz -39.83 deg; joints [46.841, -68.924, 75.776, -0.867, 83.131, 46.942]
  MoveL 123 to (129.57, 153.65, 0) mm, rotated rx 180 ry 0 rz -39.83 deg; joints [46.867, -68.924, 75.777, -0.867, 83.131, 46.967]
  MoveL 124 to (130.09, 153.67, 0) mm, rotated rx 180 ry 0 rz -39.83 deg; joints [46.893, -68.925, 75.779, -0.867, 83.131, 46.993]
  MoveL 125 to (130.82, 153.67, 0) mm, rotated rx -180 ry 0 rz -39.83 deg; joints [46.928, -68.928, 75.784, -0.867, 83.129, 47.029]
  MoveL 126 to (131.54, 153.65, 0) mm, rotated rx 180 ry 0 rz -39.83 deg; joints [46.964, -68.933, 75.792, -0.867, 83.127, 47.065]
  MoveL 127 to (132.27, 153.6, 0) mm, rotated rx 180 ry 0 rz -39.83 deg; joints [47, -68.94, 75.803, -0.867, 83.124, 47.1]
  MoveL 128 to (132.99, 153.52, 0) mm, rotated rx 180 ry 0 rz -39.83 deg; joints [47.035, -68.95, 75.817, -0.867, 83.12, 47.135]
  MoveL 129 to (133.82, 153.39, 0) mm, rotated rx -180 ry 0 rz -39.83 deg; joints [47.075, -68.965, 75.838, -0.867, 83.114, 47.176]
  MoveL 130 to (134.82, 153.18, 0) mm, rotated rx 180 ry 0 rz -39.83 deg; joints [47.124, -68.987, 75.87, -0.867, 83.105, 47.225]
  MoveL 131 to (136.19, 152.85, 0) mm, rotated rx -180 ry 0 rz -39.83 deg; joints [47.19, -69.021, 75.918, -0.867, 83.092, 47.291]
  MoveL 132 to (138.11, 152.35, 0) mm, rotated rx 180 ry 0 rz -39.83 deg; joints [47.283, -69.071, 75.989, -0.867, 83.072, 47.385]
  Establecer velocidad (1000.0 mm/s)
  MoveL 133 to (138.11, 152.35, 0) mm, rotated rx 180 ry 0 rz -39.83 deg; joints [47.283, -69.071, 75.989, -0.867, 83.072, 47.385]
  MoveL 134 to (138.11, 152.35, 20) mm, rotated rx -180 ry 0 rz -39.83 deg; joints [47.298, -69.343, 74.631, -0.864, 84.703, 47.375]
  Establecer velocidad (1000.0 mm/s)
  MoveL 135 to (65.28, 152.35, 20) mm, rotated rx 180 ry 0 rz -39.83 deg; joints [43.733, -68.85, 73.864, -0.862, 84.923, 43.806]
  MoveL 136 to (65.28, 152.35, 0) mm, rotated rx 180 ry 0 rz -39.83 deg; joints [43.719, -68.584, 75.226, -0.864, 83.294, 43.816]
  MoveL 137 to (65.28, 152.35, 0) mm, rotated rx 180 ry 0 rz -39.83 deg; joints [43.719, -68.584, 75.226, -0.864, 83.294, 43.816]
  Establecer velocidad (50.0 mm/s)
  MoveL 138 to (64.5, 152.07, 0) mm, rotated rx -180 ry 0 rz -39.83 deg; joints [43.679, -68.6, 75.248, -0.864, 83.289, 43.777]
  MoveL 139 to (63.73, 151.76, 0) mm, rotated rx 180 ry 0 rz -39.83 deg; joints [43.64, -68.619, 75.272, -0.864, 83.282, 43.738]
  MoveL 140 to (62.97, 151.43, 0) mm, rotated rx 180 ry 0 rz -39.83 deg; joints [43.601, -68.639, 75.3, -0.864, 83.275, 43.699]
  MoveL 141 to (62.23, 151.09, 0) mm, rotated rx -180 ry 0 rz -39.83 deg; joints [43.563, -68.661, 75.329, -0.864, 83.267, 43.661]
  MoveL 142 to (61.28, 150.62, 0) mm, rotated rx 180 ry 0 rz -39.83 deg; joints [43.514, -68.691, 75.369, -0.864, 83.256, 43.612]
  MoveL 143 to (60.35, 150.14, 0) mm, rotated rx 180 ry 0 rz -39.83 deg; joints [43.466, -68.723, 75.412, -0.864, 83.245, 43.564]
  MoveL 144 to (59.43, 149.63, 0) mm, rotated rx 180 ry 0 rz -39.83 deg; joints [43.418, -68.757, 75.457, -0.864, 83.233, 43.516]
  MoveL 145 to (58.51, 149.1, 0) mm, rotated rx 180 ry 0 rz -39.83 deg; joints [43.371, -68.792, 75.504, -0.864, 83.22, 43.469]
  MoveL 146 to (57.39, 148.42, 0) mm, rotated rx 180 ry 0 rz -39.83 deg; joints [43.312, -68.839, 75.566, -0.864, 83.203, 43.41]
  MoveL 147 to (56.29, 147.68, 0) mm, rotated rx 180 ry 0 rz -39.83 deg; joints [43.254, -68.89, 75.634, -0.864, 83.185, 43.353]
  MoveL 148 to (55.24, 146.89, 0) mm, rotated rx 180 ry 0 rz -39.83 deg; joints [43.198, -68.946, 75.71, -0.864, 83.165, 43.297]
  MoveL 149 to (54.27, 146.01, 0) mm, rotated rx 180 ry 0 rz -39.83 deg; joints [43.146, -69.01, 75.797, -0.864, 83.142, 43.245]
  MoveL 150 to (53.57, 145.25, 0) mm, rotated rx -180 ry 0 rz -39.83 deg; joints [43.107, -69.067, 75.873, -0.864, 83.121, 43.206]
  MoveL 151 to (52.9, 144.46, 0) mm, rotated rx 180 ry 0 rz -39.83 deg; joints [43.069, -69.127, 75.954, -0.864, 83.1, 43.169]
  MoveL 152 to (52.26, 143.64, 0) mm, rotated rx 180 ry 0 rz -39.83 deg; joints [43.033, -69.189, 76.038, -0.864, 83.077, 43.133]
  MoveL 153 to (51.61, 142.82, 0) mm, rotated rx -180 ry 0 rz -39.83 deg; joints [42.996, -69.251, 76.122, -0.864, 83.055, 43.097]
  MoveL 154 to (50.76, 141.8, 0) mm, rotated rx 180 ry 0 rz -39.83 deg; joints [42.948, -69.328, 76.226, -0.864, 83.027, 43.049]
  MoveL 155 to (49.9, 140.78, 0) mm, rotated rx 180 ry 0 rz -39.83 deg; joints [42.899, -69.404, 76.328, -0.864, 83, 43.001]
  MoveL 156 to (49.06, 139.76, 0) mm, rotated rx 180 ry 0 rz -39.83 deg; joints [42.852, -69.481, 76.432, -0.864, 82.973, 42.954]
  MoveL 157 to (48.28, 138.69, 0) mm, rotated rx -180 ry 0 rz -39.83 deg; joints [42.807, -69.562, 76.541, -0.864, 82.944, 42.909]
  MoveL 158 to (47.68, 137.74, 0) mm, rotated rx 180 ry 0 rz -39.83 deg; joints [42.772, -69.635, 76.64, -0.864, 82.918, 42.874]
  MoveL 159 to (47.13, 136.75, 0) mm, rotated rx 180 ry 0 rz -39.83 deg; joints [42.738, -69.712, 76.743, -0.864, 82.891, 42.841]
  MoveL 160 to (46.63, 135.74, 0) mm, rotated rx 180 ry 0 rz -39.83 deg; joints [42.707, -69.791, 76.85, -0.864, 82.863, 42.81]
  MoveL 161 to (46.15, 134.7, 0) mm, rotated rx 180 ry 0 rz -39.83 deg; joints [42.677, -69.873, 76.96, -0.864, 82.834, 42.781]
  MoveL 162 to (45.56, 133.33, 0) mm, rotated rx 180 ry 0 rz -39.83 deg; joints [42.639, -69.981, 77.105, -0.864, 82.796, 42.743]
  MoveL 163 to (45.02, 131.95, 0) mm, rotated rx 180 ry 0 rz -39.83 deg; joints [42.603, -70.09, 77.252, -0.864, 82.758, 42.708]
  MoveL 164 to (44.54, 130.54, 0) mm, rotated rx 180 ry 0 rz -39.83 deg; joints [42.57, -70.202, 77.403, -0.864, 82.719, 42.676]
  MoveL 165 to (44.15, 129.11, 0) mm, rotated rx 180 ry 0 rz -39.83 deg; joints [42.542, -70.317, 77.557, -0.864, 82.679, 42.648]
  MoveL 166 to (43.9, 127.9, 0) mm, rotated rx -180 ry 0 rz -39.83 deg; joints [42.521, -70.416, 77.689, -0.864, 82.645, 42.628]
  MoveL 167 to (43.72, 126.67, 0) mm, rotated rx 180 ry 0 rz -39.83 deg; joints [42.504, -70.516, 77.824, -0.864, 82.611, 42.611]
  MoveL 168 to (43.58, 125.43, 0) mm, rotated rx 180 ry 0 rz -39.83 deg; joints [42.489, -70.617, 77.96, -0.864, 82.576, 42.597]
  MoveL 169 to (43.49, 124.19, 0) mm, rotated rx 180 ry 0 rz -39.83 deg; joints [42.476, -70.72, 78.097, -0.864, 82.541, 42.584]
  MoveL 170 to (43.43, 123.02, 0) mm, rotated rx -180 ry 0 rz -39.83 deg; joints [42.465, -70.816, 78.226, -0.864, 82.508, 42.574]
  MoveL 171 to (43.4, 121.86, 0) mm, rotated rx 180 ry 0 rz -39.83 deg; joints [42.456, -70.913, 78.355, -0.864, 82.476, 42.566]
  MoveL 172 to (43.42, 120.69, 0) mm, rotated rx 180 ry 0 rz -39.83 deg; joints [42.449, -71.009, 78.484, -0.864, 82.443, 42.559]
  MoveL 173 to (43.49, 119.53, 0) mm, rotated rx 180 ry 0 rz -39.83 deg; joints [42.445, -71.106, 78.614, -0.864, 82.411, 42.555]
  MoveL 174 to (43.68, 117.85, 0) mm, rotated rx 180 ry 0 rz -39.83 deg; joints [42.443, -71.248, 78.803, -0.864, 82.363, 42.554]
  MoveL 175 to (43.97, 116.18, 0) mm, rotated rx 180 ry 0 rz -39.83 deg; joints [42.446, -71.39, 78.992, -0.864, 82.316, 42.558]
  MoveL 176 to (44.36, 114.52, 0) mm, rotated rx 180 ry 0 rz -39.83 deg; joints [42.454, -71.531, 79.18, -0.864, 82.27, 42.567]
  MoveL 177 to (44.82, 112.88, 0) mm, rotated rx -180 ry 0 rz -39.83 deg; joints [42.466, -71.673, 79.368, -0.865, 82.223, 42.579]
  MoveL 178 to (45.27, 111.47, 0) mm, rotated rx 180 ry 0 rz -39.83 deg; joints [42.479, -71.795, 79.53, -0.865, 82.183, 42.593]
  MoveL 179 to (45.79, 110.08, 0) mm, rotated rx 180 ry 0 rz -39.83 deg; joints [42.496, -71.915, 79.69, -0.865, 82.144, 42.61]
  MoveL 180 to (46.38, 108.73, 0) mm, rotated rx 180 ry 0 rz -39.83 deg; joints [42.517, -72.034, 79.846, -0.865, 82.106, 42.632]
  MoveL 181 to (47.08, 107.43, 0) mm, rotated rx 180 ry 0 rz -39.83 deg; joints [42.543, -72.149, 79.999, -0.865, 82.069, 42.658]
  MoveL 182 to (48.05, 105.97, 0) mm, rotated rx 180 ry 0 rz -39.83 deg; joints [42.582, -72.279, 80.171, -0.865, 82.028, 42.698]
  MoveL 183 to (49.16, 104.62, 0) mm, rotated rx 180 ry 0 rz -39.83 deg; joints [42.629, -72.403, 80.335, -0.865, 81.988, 42.746]
  MoveL 184 to (50.4, 103.37, 0) mm, rotated rx 180 ry 0 rz -39.83 deg; joints [42.683, -72.519, 80.489, -0.865, 81.951, 42.801]
  MoveL 185 to (51.74, 102.24, 0) mm, rotated rx 180 ry 0 rz -39.83 deg; joints [42.744, -72.627, 80.632, -0.866, 81.917, 42.862]
  MoveL 186 to (52.99, 101.33, 0) mm, rotated rx -180 ry 0 rz -39.83 deg; joints [42.801, -72.715, 80.748, -0.866, 81.889, 42.92]
  MoveL 187 to (54.3, 100.52, 0) mm, rotated rx -180 ry 0 rz -39.83 deg; joints [42.862, -72.795, 80.855, -0.866, 81.864, 42.981]
  MoveL 188 to (55.67, 99.8, 0) mm, rotated rx 180 ry 0 rz -39.83 deg; joints [42.927, -72.868, 80.953, -0.866, 81.841, 43.046]
  MoveL 189 to (57.07, 99.18, 0) mm, rotated rx 180 ry 0 rz -39.83 deg; joints [42.994, -72.934, 81.041, -0.866, 81.82, 43.114]
  MoveL 190 to (58.3, 98.71, 0) mm, rotated rx 180 ry 0 rz -39.83 deg; joints [43.054, -72.985, 81.108, -0.866, 81.804, 43.174]
  MoveL 191 to (59.56, 98.32, 0) mm, rotated rx 180 ry 0 rz -39.83 deg; joints [43.115, -73.03, 81.169, -0.866, 81.79, 43.235]
  MoveL 192 to (60.84, 97.98, 0) mm, rotated rx 180 ry 0 rz -39.83 deg; joints [43.178, -73.071, 81.223, -0.867, 81.777, 43.298]
  MoveL 193 to (62.13, 97.71, 0) mm, rotated rx 180 ry 0 rz -39.83 deg; joints [43.242, -73.106, 81.27, -0.867, 81.766, 43.363]
  MoveL 194 to (63.62, 97.48, 0) mm, rotated rx 180 ry 0 rz -39.83 deg; joints [43.317, -73.139, 81.316, -0.867, 81.755, 43.438]
  MoveL 195 to (65.12, 97.33, 0) mm, rotated rx 180 ry 0 rz -39.83 deg; joints [43.392, -73.166, 81.352, -0.867, 81.746, 43.513]
  MoveL 196 to (66.62, 97.27, 0) mm, rotated rx 180 ry 0 rz -39.83 deg; joints [43.469, -73.185, 81.379, -0.867, 81.739, 43.59]
  MoveL 197 to (68.12, 97.31, 0) mm, rotated rx 180 ry 0 rz -39.83 deg; joints [43.546, -73.196, 81.395, -0.867, 81.735, 43.667]
  MoveL 198 to (69.57, 97.45, 0) mm, rotated rx -180 ry 0 rz -39.83 deg; joints [43.621, -73.198, 81.4, -0.867, 81.734, 43.742]
  MoveL 199 to (71.01, 97.68, 0) mm, rotated rx 180 ry 0 rz -39.83 deg; joints [43.695, -73.192, 81.394, -0.867, 81.735, 43.816]
  MoveL 200 to (72.44, 97.99, 0) mm, rotated rx 180 ry 0 rz -39.83 deg; joints [43.77, -73.18, 81.38, -0.867, 81.738, 43.891]
  MoveL 201 to (73.85, 98.38, 0) mm, rotated rx 180 ry 0 rz -39.83 deg; joints [43.844, -73.16, 81.356, -0.867, 81.743, 43.965]
  MoveL 202 to (75.02, 98.76, 0) mm, rotated rx -180 ry 0 rz -39.83 deg; joints [43.906, -73.139, 81.33, -0.867, 81.749, 44.027]
  MoveL 203 to (76.17, 99.19, 0) mm, rotated rx -180 ry 0 rz -39.83 deg; joints [43.967, -73.113, 81.298, -0.867, 81.756, 44.088]
  MoveL 204 to (77.29, 99.69, 0) mm, rotated rx 180 ry 0 rz -39.83 deg; joints [44.027, -73.082, 81.26, -0.868, 81.764, 44.148]
  MoveL 205 to (78.38, 100.24, 0) mm, rotated rx 180 ry 0 rz -39.83 deg; joints [44.086, -73.046, 81.214, -0.868, 81.775, 44.206]
  MoveL 206 to (79.78, 101.09, 0) mm, rotated rx 180 ry 0 rz -39.83 deg; joints [44.162, -72.988, 81.14, -0.868, 81.791, 44.282]
  MoveL 207 to (81.13, 102.03, 0) mm, rotated rx -180 ry 0 rz -39.83 deg; joints [44.236, -72.922, 81.056, -0.868, 81.811, 44.356]
  MoveL 208 to (82.44, 103.04, 0) mm, rotated rx 180 ry 0 rz -39.83 deg; joints [44.308, -72.849, 80.962, -0.868, 81.832, 44.427]
  MoveL 209 to (83.7, 104.1, 0) mm, rotated rx 180 ry 0 rz -39.83 deg; joints [44.378, -72.771, 80.863, -0.868, 81.855, 44.497]
  MoveL 210 to (85.05, 105.29, 0) mm, rotated rx -180 ry 0 rz -39.83 deg; joints [44.452, -72.684, 80.75, -0.868, 81.881, 44.571]
  MoveL 211 to (86.35, 106.52, 0) mm, rotated rx -180 ry 0 rz -39.83 deg; joints [44.525, -72.592, 80.632, -0.868, 81.909, 44.643]
  MoveL 212 to (87.6, 107.81, 0) mm, rotated rx -180 ry 0 rz -39.83 deg; joints [44.594, -72.496, 80.507, -0.868, 81.938, 44.712]
  MoveL 213 to (88.77, 109.16, 0) mm, rotated rx -180 ry 0 rz -39.83 deg; joints [44.66, -72.393, 80.374, -0.868, 81.97, 44.778]
  MoveL 214 to (89.65, 110.29, 0) mm, rotated rx 180 ry 0 rz -39.83 deg; joints [44.71, -72.305, 80.261, -0.868, 81.997, 44.828]
  MoveL 215 to (90.47, 111.47, 0) mm, rotated rx -180 ry 0 rz -39.83 deg; joints [44.758, -72.214, 80.141, -0.868, 82.025, 44.875]
  MoveL 216 to (91.24, 112.69, 0) mm, rotated rx 180 ry 0 rz -39.83 deg; joints [44.803, -72.118, 80.017, -0.868, 82.055, 44.919]
  MoveL 217 to (91.96, 113.95, 0) mm, rotated rx 180 ry 0 rz -39.83 deg; joints [44.845, -72.02, 79.888, -0.868, 82.086, 44.961]
  MoveL 218 to (92.79, 115.55, 0) mm, rotated rx 180 ry 0 rz -39.83 deg; joints [44.895, -71.893, 79.721, -0.868, 82.126, 45.01]
  MoveL 219 to (93.54, 117.2, 0) mm, rotated rx -180 ry 0 rz -39.83 deg; joints [44.94, -71.761, 79.549, -0.868, 82.168, 45.054]
  MoveL 220 to (94.19, 118.88, 0) mm, rotated rx 180 ry 0 rz -39.83 deg; joints [44.981, -71.626, 79.371, -0.867, 82.211, 45.095]
  MoveL 221 to (94.76, 120.6, 0) mm, rotated rx 180 ry 0 rz -39.83 deg; joints [45.017, -71.487, 79.188, -0.867, 82.256, 45.13]
  MoveL 222 to (95.27, 122.52, 0) mm, rotated rx -180 ry 0 rz -39.83 deg; joints [45.051, -71.331, 78.98, -0.867, 82.308, 45.164]
  MoveL 223 to (95.66, 124.48, 0) mm, rotated rx -180 ry 0 rz -39.83 deg; joints [45.079, -71.171, 78.768, -0.867, 82.36, 45.191]
  MoveL 224 to (95.93, 126.46, 0) mm, rotated rx 180 ry 0 rz -39.83 deg; joints [45.102, -71.008, 78.551, -0.867, 82.415, 45.213]
  MoveL 225 to (96.09, 128.45, 0) mm, rotated rx 180 ry 0 rz -39.83 deg; joints [45.119, -70.843, 78.33, -0.867, 82.47, 45.229]
  MoveL 226 to (96.13, 129.89, 0) mm, rotated rx -180 ry 0 rz -39.83 deg; joints [45.127, -70.723, 78.17, -0.867, 82.511, 45.237]
  MoveL 227 to (96.11, 131.32, 0) mm, rotated rx 180 ry 0 rz -39.83 deg; joints [45.132, -70.603, 78.009, -0.867, 82.552, 45.241]
  MoveL 228 to (96.01, 132.75, 0) mm, rotated rx 180 ry 0 rz -39.83 deg; joints [45.134, -70.483, 77.847, -0.867, 82.593, 45.242]
  MoveL 229 to (95.82, 134.17, 0) mm, rotated rx 180 ry 0 rz -39.83 deg; joints [45.131, -70.362, 77.686, -0.867, 82.635, 45.238]
  MoveL 230 to (95.51, 135.74, 0) mm, rotated rx 180 ry 0 rz -39.83 deg; joints [45.122, -70.229, 77.506, -0.867, 82.681, 45.229]
  MoveL 231 to (95.09, 137.28, 0) mm, rotated rx 180 ry 0 rz -39.83 deg; joints [45.108, -70.097, 77.326, -0.867, 82.728, 45.214]
  MoveL 232 to (94.57, 138.8, 0) mm, rotated rx -180 ry 0 rz -39.83 deg; joints [45.089, -69.966, 77.149, -0.866, 82.774, 45.194]
  MoveL 233 to (93.96, 140.29, 0) mm, rotated rx 180 ry 0 rz -39.83 deg; joints [45.065, -69.836, 76.973, -0.866, 82.82, 45.17]
  MoveL 234 to (93.12, 142.02, 0) mm, rotated rx 180 ry 0 rz -39.83 deg; joints [45.032, -69.685, 76.767, -0.866, 82.875, 45.135]
  MoveL 235 to (92.16, 143.67, 0) mm, rotated rx -180 ry 0 rz -39.83 deg; joints [44.992, -69.539, 76.567, -0.866, 82.928, 45.095]
  MoveL 236 to (91.07, 145.24, 0) mm, rotated rx 180 ry 0 rz -39.83 deg; joints [44.945, -69.399, 76.376, -0.866, 82.979, 45.047]
  MoveL 237 to (89.83, 146.68, 0) mm, rotated rx 180 ry 0 rz -39.83 deg; joints [44.89, -69.269, 76.196, -0.866, 83.027, 44.992]
  MoveL 238 to (88.97, 147.52, 0) mm, rotated rx 180 ry 0 rz -39.83 deg; joints [44.852, -69.191, 76.09, -0.866, 83.056, 44.953]
  MoveL 239 to (88.05, 148.31, 0) mm, rotated rx -180 ry 0 rz -39.83 deg; joints [44.811, -69.118, 75.988, -0.866, 83.083, 44.911]
  MoveL 240 to (87.09, 149.04, 0) mm, rotated rx 180 ry 0 rz -39.83 deg; joints [44.767, -69.049, 75.892, -0.866, 83.109, 44.867]
  MoveL 241 to (86.1, 149.74, 0) mm, rotated rx 180 ry 0 rz -39.83 deg; joints [44.722, -68.982, 75.8, -0.865, 83.134, 44.822]
  MoveL 242 to (85.17, 150.33, 0) mm, rotated rx 180 ry 0 rz -39.83 deg; joints [44.679, -68.925, 75.72, -0.865, 83.156, 44.778]
  MoveL 243 to (84.22, 150.89, 0) mm, rotated rx 180 ry 0 rz -39.83 deg; joints [44.635, -68.87, 75.644, -0.865, 83.177, 44.734]
  MoveL 244 to (83.24, 151.4, 0) mm, rotated rx -180 ry 0 rz -39.83 deg; joints [44.59, -68.819, 75.573, -0.865, 83.196, 44.689]
  MoveL 245 to (82.24, 151.87, 0) mm, rotated rx 180 ry 0 rz -39.83 deg; joints [44.543, -68.772, 75.507, -0.865, 83.214, 44.642]
  MoveL 246 to (81.33, 152.23, 0) mm, rotated rx -180 ry 0 rz -39.83 deg; joints [44.5, -68.734, 75.454, -0.865, 83.229, 44.599]
  MoveL 247 to (80.4, 152.55, 0) mm, rotated rx 180 ry 0 rz -39.83 deg; joints [44.457, -68.699, 75.405, -0.865, 83.242, 44.555]
  MoveL 248 to (79.46, 152.83, 0) mm, rotated rx 180 ry 0 rz -39.83 deg; joints [44.412, -68.668, 75.361, -0.865, 83.255, 44.51]
  MoveL 249 to (78.51, 153.06, 0) mm, rotated rx 180 ry 0 rz -39.83 deg; joints [44.367, -68.641, 75.322, -0.865, 83.265, 44.465]
  MoveL 250 to (77.73, 153.22, 0) mm, rotated rx 180 ry 0 rz -39.83 deg; joints [44.33, -68.621, 75.294, -0.865, 83.273, 44.427]
  MoveL 251 to (76.95, 153.34, 0) mm, rotated rx 180 ry 0 rz -39.83 deg; joints [44.292, -68.604, 75.269, -0.865, 83.28, 44.39]
  MoveL 252 to (76.17, 153.45, 0) mm, rotated rx 180 ry 0 rz -39.83 deg; joints [44.255, -68.588, 75.247, -0.865, 83.286, 44.352]
  MoveL 253 to (75.38, 153.53, 0) mm, rotated rx 180 ry 0 rz -39.83 deg; joints [44.217, -68.574, 75.227, -0.865, 83.292, 44.314]
  MoveL 254 to (74.86, 153.58, 0) mm, rotated rx 180 ry 0 rz -39.83 deg; joints [44.192, -68.566, 75.214, -0.865, 83.296, 44.289]
  MoveL 255 to (74.34, 153.62, 0) mm, rotated rx 180 ry 0 rz -39.83 deg; joints [44.167, -68.558, 75.203, -0.865, 83.299, 44.264]
  MoveL 256 to (73.82, 153.65, 0) mm, rotated rx -180 ry 0 rz -39.83 deg; joints [44.141, -68.551, 75.193, -0.865, 83.302, 44.239]
  MoveL 257 to (73.3, 153.67, 0) mm, rotated rx -180 ry 0 rz -39.83 deg; joints [44.116, -68.545, 75.184, -0.865, 83.304, 44.213]
  MoveL 258 to (72.57, 153.67, 0) mm, rotated rx 180 ry 0 rz -39.83 deg; joints [44.081, -68.538, 75.173, -0.865, 83.307, 44.178]
  MoveL 259 to (71.85, 153.65, 0) mm, rotated rx 180 ry 0 rz -39.83 deg; joints [44.045, -68.534, 75.166, -0.864, 83.309, 44.142]
  MoveL 260 to (71.12, 153.6, 0) mm, rotated rx 180 ry 0 rz -39.83 deg; joints [44.01, -68.531, 75.162, -0.864, 83.311, 44.107]
  MoveL 261 to (70.4, 153.52, 0) mm, rotated rx -180 ry 0 rz -39.83 deg; joints [43.974, -68.531, 75.161, -0.864, 83.311, 44.071]
  MoveL 262 to (69.57, 153.39, 0) mm, rotated rx -180 ry 0 rz -39.83 deg; joints [43.933, -68.535, 75.165, -0.864, 83.31, 44.03]
  MoveL 263 to (68.57, 153.18, 0) mm, rotated rx 180 ry 0 rz -39.83 deg; joints [43.883, -68.544, 75.175, -0.864, 83.307, 43.98]
  MoveL 264 to (67.2, 152.85, 0) mm, rotated rx 180 ry 0 rz -39.83 deg; joints [43.815, -68.559, 75.195, -0.864, 83.302, 43.912]
  MoveL 265 to (65.28, 152.35, 0) mm, rotated rx 180 ry 0 rz -39.83 deg; joints [43.719, -68.584, 75.226, -0.864, 83.294, 43.816]
  Establecer velocidad (1000.0 mm/s)
  MoveL 266 to (65.28, 152.35, 0) mm, rotated rx 180 ry 0 rz -39.83 deg; joints [43.719, -68.584, 75.226, -0.864, 83.294, 43.816]
  MoveL 267 to (65.28, 152.35, 20) mm, rotated rx 180 ry 0 rz -39.83 deg; joints [43.733, -68.85, 73.864, -0.862, 84.923, 43.806]
  Establecer velocidad (1000.0 mm/s)
  MoveL 268 to (71.43, 178.24, 20) mm, rotated rx 180 ry 0 rz -39.83 deg; joints [44.166, -66.684, 70.869, -0.861, 85.758, 44.226]
  MoveL 269 to (71.43, 178.24, 0) mm, rotated rx -180 ry 0 rz -39.83 deg; joints [44.151, -66.44, 72.249, -0.863, 84.133, 44.236]
  MoveL 270 to (71.43, 178.24, 0) mm, rotated rx -180 ry 0 rz -39.83 deg; joints [44.151, -66.44, 72.249, -0.863, 84.133, 44.236]
  Establecer velocidad (50.0 mm/s)
  MoveL 271 to (71.48, 178.2, 0) mm, rotated rx -180 ry 0 rz -39.83 deg; joints [44.154, -66.443, 72.255, -0.863, 84.132, 44.238]
  MoveL 272 to (71.54, 178.16, 0) mm, rotated rx 180 ry 0 rz -39.83 deg; joints [44.156, -66.447, 72.26, -0.863, 84.13, 44.241]
  MoveL 273 to (71.58, 178.12, 0) mm, rotated rx 180 ry 0 rz -39.83 deg; joints [44.158, -66.451, 72.266, -0.863, 84.129, 44.243]
  MoveL 274 to (71.61, 178.07, 0) mm, rotated rx -180 ry 0 rz -39.83 deg; joints [44.159, -66.456, 72.273, -0.863, 84.127, 44.244]
  MoveL 275 to (71.65, 177.98, 0) mm, rotated rx -180 ry 0 rz -39.83 deg; joints [44.16, -66.464, 72.285, -0.863, 84.123, 44.245]
  MoveL 276 to (71.65, 177.87, 0) mm, rotated rx -180 ry 0 rz -39.83 deg; joints [44.16, -66.474, 72.298, -0.863, 84.119, 44.245]
  MoveL 277 to (71.63, 177.75, 0) mm, rotated rx 180 ry 0 rz -39.83 deg; joints [44.159, -66.484, 72.312, -0.863, 84.115, 44.243]
  MoveL 278 to (71.61, 177.63, 0) mm, rotated rx 180 ry 0 rz -39.83 deg; joints [44.157, -66.493, 72.325, -0.863, 84.111, 44.242]
  MoveL 279 to (71.58, 177.5, 0) mm, rotated rx 180 ry 0 rz -39.83 deg; joints [44.155, -66.505, 72.341, -0.863, 84.107, 44.24]
  MoveL 280 to (71.56, 177.37, 0) mm, rotated rx 180 ry 0 rz -39.83 deg; joints [44.153, -66.515, 72.356, -0.863, 84.102, 44.238]
  MoveL 281 to (71.53, 177.25, 0) mm, rotated rx 180 ry 0 rz -39.83 deg; joints [44.151, -66.526, 72.371, -0.863, 84.098, 44.236]
  MoveL 282 to (71.49, 177.12, 0) mm, rotated rx 180 ry 0 rz -39.83 deg; joints [44.149, -66.536, 72.385, -0.863, 84.094, 44.234]
  MoveL 283 to (71.43, 176.92, 0) mm, rotated rx 180 ry 0 rz -39.83 deg; joints [44.144, -66.553, 72.409, -0.863, 84.087, 44.23]
  MoveL 284 to (71.35, 176.72, 0) mm, rotated rx 180 ry 0 rz -39.83 deg; joints [44.14, -66.569, 72.432, -0.863, 84.08, 44.225]
  MoveL 285 to (71.26, 176.52, 0) mm, rotated rx 180 ry 0 rz -39.83 deg; joints [44.135, -66.586, 72.455, -0.863, 84.074, 44.22]
  MoveL 286 to (71.17, 176.32, 0) mm, rotated rx -180 ry 0 rz -39.83 deg; joints [44.129, -66.602, 72.477, -0.863, 84.067, 44.215]
  MoveL 287 to (71.01, 176.01, 0) mm, rotated rx 180 ry 0 rz -39.83 deg; joints [44.12, -66.627, 72.513, -0.863, 84.057, 44.206]
  MoveL 288 to (70.84, 175.7, 0) mm, rotated rx 180 ry 0 rz -39.83 deg; joints [44.11, -66.652, 72.548, -0.863, 84.047, 44.196]
  MoveL 289 to (70.66, 175.4, 0) mm, rotated rx -180 ry 0 rz -39.83 deg; joints [44.1, -66.676, 72.581, -0.863, 84.037, 44.186]
  MoveL 290 to (70.47, 175.1, 0) mm, rotated rx -180 ry 0 rz -39.83 deg; joints [44.089, -66.7, 72.614, -0.863, 84.028, 44.176]
  MoveL 291 to (69.99, 174.43, 0) mm, rotated rx -180 ry 0 rz -39.83 deg; joints [44.063, -66.753, 72.688, -0.863, 84.007, 44.15]
  MoveL 292 to (69.49, 173.78, 0) mm, rotated rx 180 ry 0 rz -39.83 deg; joints [44.036, -66.804, 72.759, -0.863, 83.986, 44.123]
  MoveL 293 to (68.96, 173.14, 0) mm, rotated rx 180 ry 0 rz -39.83 deg; joints [44.007, -66.854, 72.828, -0.863, 83.966, 44.094]
  MoveL 294 to (68.42, 172.52, 0) mm, rotated rx 180 ry 0 rz -39.83 deg; joints [43.978, -66.902, 72.896, -0.863, 83.947, 44.066]
  MoveL 295 to (67.07, 170.96, 0) mm, rotated rx 180 ry 0 rz -39.83 deg; joints [43.905, -67.022, 73.062, -0.863, 83.9, 43.993]
  MoveL 296 to (65.69, 169.43, 0) mm, rotated rx 180 ry 0 rz -39.83 deg; joints [43.831, -67.14, 73.225, -0.863, 83.853, 43.92]
  MoveL 297 to (64.29, 167.93, 0) mm, rotated rx 180 ry 0 rz -39.83 deg; joints [43.756, -67.255, 73.384, -0.863, 83.808, 43.845]
  MoveL 298 to (62.85, 166.46, 0) mm, rotated rx 180 ry 0 rz -39.83 deg; joints [43.679, -67.366, 73.537, -0.863, 83.765, 43.769]
  MoveL 299 to (61.26, 164.94, 0) mm, rotated rx 180 ry 0 rz -39.83 deg; joints [43.594, -67.48, 73.694, -0.863, 83.721, 43.684]
  MoveL 300 to (59.63, 163.45, 0) mm, rotated rx -180 ry 0 rz -39.83 deg; joints [43.507, -67.591, 73.846, -0.863, 83.679, 43.598]
  MoveL 301 to (57.97, 161.99, 0) mm, rotated rx 180 ry 0 rz -39.83 deg; joints [43.419, -67.699, 73.994, -0.863, 83.637, 43.511]
  MoveL 302 to (56.3, 160.53, 0) mm, rotated rx 180 ry 0 rz -39.83 deg; joints [43.33, -67.806, 74.14, -0.863, 83.597, 43.422]
  MoveL 303 to (54.03, 158.54, 0) mm, rotated rx 180 ry 0 rz -39.83 deg; joints [43.208, -67.951, 74.339, -0.863, 83.542, 43.302]
  MoveL 304 to (51.74, 156.58, 0) mm, rotated rx 180 ry 0 rz -39.83 deg; joints [43.086, -68.094, 74.533, -0.863, 83.488, 43.18]
  MoveL 305 to (49.4, 154.69, 0) mm, rotated rx -180 ry 0 rz -39.83 deg; joints [42.961, -68.229, 74.717, -0.863, 83.437, 43.056]
  MoveL 306 to (46.99, 152.9, 0) mm, rotated rx -180 ry 0 rz -39.83 deg; joints [42.833, -68.355, 74.887, -0.863, 83.391, 42.929]
  MoveL 307 to (45.38, 151.81, 0) mm, rotated rx -180 ry 0 rz -39.83 deg; joints [42.749, -68.429, 74.988, -0.863, 83.364, 42.845]
  MoveL 308 to (43.74, 150.76, 0) mm, rotated rx 180 ry 0 rz -39.83 deg; joints [42.663, -68.5, 75.083, -0.863, 83.338, 42.759]
  MoveL 309 to (42.1, 149.72, 0) mm, rotated rx 180 ry 0 rz -39.83 deg; joints [42.576, -68.569, 75.176, -0.863, 83.313, 42.673]
  MoveL 310 to (40.46, 148.68, 0) mm, rotated rx 180 ry 0 rz -39.83 deg; joints [42.49, -68.639, 75.27, -0.863, 83.288, 42.587]
  MoveL 311 to (39.41, 148, 0) mm, rotated rx 180 ry 0 rz -39.83 deg; joints [42.435, -68.684, 75.331, -0.863, 83.271, 42.532]
  MoveL 312 to (38.36, 147.34, 0) mm, rotated rx 180 ry 0 rz -39.83 deg; joints [42.379, -68.728, 75.39, -0.862, 83.255, 42.477]
  MoveL 313 to (37.29, 146.72, 0) mm, rotated rx -180 ry 0 rz -39.83 deg; joints [42.323, -68.768, 75.442, -0.862, 83.241, 42.42]
  MoveL 314 to (36.17, 146.19, 0) mm, rotated rx -180 ry 0 rz -39.83 deg; joints [42.265, -68.8, 75.485, -0.862, 83.23, 42.363]
  MoveL 315 to (35.75, 146.01, 0) mm, rotated rx -180 ry 0 rz -39.83 deg; joints [42.243, -68.81, 75.498, -0.862, 83.227, 42.341]
  MoveL 316 to (35.33, 145.86, 0) mm, rotated rx 180 ry 0 rz -39.83 deg; joints [42.222, -68.818, 75.509, -0.862, 83.224, 42.32]
  MoveL 317 to (34.9, 145.71, 0) mm, rotated rx 180 ry 0 rz -39.83 deg; joints [42.2, -68.825, 75.518, -0.862, 83.221, 42.298]
  MoveL 318 to (34.47, 145.57, 0) mm, rotated rx -180 ry 0 rz -39.83 deg; joints [42.178, -68.832, 75.527, -0.862, 83.219, 42.276]
  MoveL 319 to (34.15, 145.48, 0) mm, rotated rx 180 ry 0 rz -39.83 deg; joints [42.162, -68.836, 75.532, -0.862, 83.218, 42.26]
  MoveL 320 to (33.82, 145.4, 0) mm, rotated rx 180 ry 0 rz -39.83 deg; joints [42.145, -68.839, 75.535, -0.862, 83.217, 42.243]
  MoveL 321 to (33.48, 145.34, 0) mm, rotated rx 180 ry 0 rz -39.83 deg; joints [42.128, -68.84, 75.536, -0.862, 83.217, 42.226]
  MoveL 322 to (33.13, 145.32, 0) mm, rotated rx 180 ry 0 rz -39.83 deg; joints [42.111, -68.838, 75.533, -0.862, 83.218, 42.209]
  MoveL 323 to (32.91, 145.33, 0) mm, rotated rx 180 ry 0 rz -39.83 deg; joints [42.101, -68.834, 75.528, -0.862, 83.219, 42.199]
  MoveL 324 to (32.7, 145.36, 0) mm, rotated rx 180 ry 0 rz -39.83 deg; joints [42.091, -68.829, 75.521, -0.862, 83.221, 42.188]
  MoveL 325 to (32.5, 145.42, 0) mm, rotated rx 180 ry 0 rz -39.83 deg; joints [42.081, -68.822, 75.51, -0.862, 83.224, 42.179]
  MoveL 326 to (32.33, 145.52, 0) mm, rotated rx 180 ry 0 rz -39.83 deg; joints [42.074, -68.811, 75.495, -0.862, 83.228, 42.172]
  MoveL 327 to (32.25, 145.61, 0) mm, rotated rx 180 ry 0 rz -39.83 deg; joints [42.07, -68.803, 75.485, -0.862, 83.231, 42.168]
  MoveL 328 to (32.18, 145.7, 0) mm, rotated rx 180 ry 0 rz -39.83 deg; joints [42.067, -68.794, 75.472, -0.862, 83.234, 42.165]
  MoveL 329 to (32.11, 145.8, 0) mm, rotated rx 180 ry 0 rz -39.83 deg; joints [42.065, -68.785, 75.459, -0.862, 83.238, 42.163]
  MoveL 330 to (32.05, 145.91, 0) mm, rotated rx -180 ry 0 rz -39.83 deg; joints [42.063, -68.775, 75.446, -0.862, 83.241, 42.16]
  MoveL 331 to (32.05, 145.91, 0) mm, rotated rx -180 ry 0 rz -39.83 deg; joints [42.063, -68.775, 75.446, -0.862, 83.241, 42.16]
  MoveL 332 to (31.99, 146.46, 0) mm, rotated rx 180 ry 0 rz -39.83 deg; joints [42.064, -68.728, 75.381, -0.862, 83.259, 42.161]
  MoveL 333 to (31.94, 147.01, 0) mm, rotated rx 180 ry 0 rz -39.83 deg; joints [42.065, -68.682, 75.317, -0.862, 83.277, 42.162]
  MoveL 334 to (31.9, 147.56, 0) mm, rotated rx 180 ry 0 rz -39.83 deg; joints [42.067, -68.635, 75.253, -0.862, 83.294, 42.164]
  MoveL 335 to (31.87, 148.11, 0) mm, rotated rx 180 ry 0 rz -39.83 deg; joints [42.069, -68.588, 75.189, -0.862, 83.312, 42.166]
  MoveL 336 to (31.86, 149.49, 0) mm, rotated rx 180 ry 0 rz -39.83 deg; joints [42.078, -68.473, 75.03, -0.862, 83.355, 42.174]
  MoveL 337 to (31.93, 150.86, 0) mm, rotated rx -180 ry 0 rz -39.83 deg; joints [42.091, -68.358, 74.872, -0.862, 83.399, 42.187]
  MoveL 338 to (32.07, 152.23, 0) mm, rotated rx 180 ry 0 rz -39.83 deg; joints [42.107, -68.244, 74.715, -0.862, 83.442, 42.202]
  MoveL 339 to (32.26, 153.6, 0) mm, rotated rx 180 ry 0 rz -39.83 deg; joints [42.126, -68.131, 74.559, -0.862, 83.485, 42.22]
  MoveL 340 to (32.46, 154.79, 0) mm, rotated rx 180 ry 0 rz -39.83 deg; joints [42.144, -68.033, 74.424, -0.862, 83.522, 42.237]
  MoveL 341 to (32.7, 155.98, 0) mm, rotated rx 180 ry 0 rz -39.83 deg; joints [42.163, -67.936, 74.289, -0.862, 83.56, 42.256]
  MoveL 342 to (32.98, 157.15, 0) mm, rotated rx 180 ry 0 rz -39.83 deg; joints [42.184, -67.84, 74.157, -0.862, 83.597, 42.277]
  MoveL 343 to (33.3, 158.31, 0) mm, rotated rx 180 ry 0 rz -39.83 deg; joints [42.208, -67.746, 74.027, -0.862, 83.633, 42.3]
  MoveL 344 to (33.61, 159.26, 0) mm, rotated rx 180 ry 0 rz -39.83 deg; joints [42.229, -67.669, 73.921, -0.862, 83.663, 42.32]
  MoveL 345 to (33.95, 160.19, 0) mm, rotated rx 180 ry 0 rz -39.83 deg; joints [42.252, -67.594, 73.817, -0.862, 83.692, 42.342]
  MoveL 346 to (34.32, 161.11, 0) mm, rotated rx 180 ry 0 rz -39.83 deg; joints [42.276, -67.52, 73.715, -0.862, 83.721, 42.366]
  MoveL 347 to (34.73, 162.02, 0) mm, rotated rx 180 ry 0 rz -39.83 deg; joints [42.301, -67.448, 73.614, -0.862, 83.749, 42.391]
  MoveL 348 to (35.07, 162.73, 0) mm, rotated rx 180 ry 0 rz -39.83 deg; joints [42.322, -67.392, 73.537, -0.862, 83.771, 42.412]
  MoveL 349 to (35.43, 163.43, 0) mm, rotated rx 180 ry 0 rz -39.83 deg; joints [42.344, -67.337, 73.461, -0.862, 83.792, 42.433]
  MoveL 350 to (35.81, 164.11, 0) mm, rotated rx -180 ry 0 rz -39.83 deg; joints [42.367, -67.283, 73.386, -0.862, 83.814, 42.456]
  MoveL 351 to (36.21, 164.79, 0) mm, rotated rx 180 ry 0 rz -39.83 deg; joints [42.39, -67.23, 73.313, -0.862, 83.834, 42.479]
  MoveL 352 to (36.79, 165.69, 0) mm, rotated rx -180 ry 0 rz -39.83 deg; joints [42.424, -67.16, 73.216, -0.862, 83.862, 42.512]
  MoveL 353 to (37.4, 166.57, 0) mm, rotated rx -180 ry 0 rz -39.83 deg; joints [42.459, -67.092, 73.122, -0.862, 83.889, 42.547]
  MoveL 354 to (38.04, 167.43, 0) mm, rotated rx 180 ry 0 rz -39.83 deg; joints [42.495, -67.027, 73.031, -0.862, 83.915, 42.583]
  MoveL 355 to (38.71, 168.26, 0) mm, rotated rx 180 ry 0 rz -39.83 deg; joints [42.533, -66.963, 72.943, -0.862, 83.94, 42.62]
  MoveL 356 to (39.42, 169.08, 0) mm, rotated rx -180 ry 0 rz -39.83 deg; joints [42.571, -66.902, 72.857, -0.862, 83.964, 42.658]
  MoveL 357 to (40.14, 169.87, 0) mm, rotated rx 180 ry 0 rz -39.83 deg; joints [42.611, -66.842, 72.775, -0.862, 83.988, 42.698]
  MoveL 358 to (40.89, 170.65, 0) mm, rotated rx 180 ry 0 rz -39.83 deg; joints [42.652, -66.784, 72.695, -0.862, 84.011, 42.738]
  MoveL 359 to (41.65, 171.41, 0) mm, rotated rx 180 ry 0 rz -39.83 deg; joints [42.693, -66.728, 72.616, -0.862, 84.033, 42.779]
  MoveL 360 to (42.47, 172.2, 0) mm, rotated rx -180 ry 0 rz -39.83 deg; joints [42.737, -66.67, 72.535, -0.862, 84.056, 42.822]
  MoveL 361 to (43.3, 172.96, 0) mm, rotated rx 180 ry 0 rz -39.83 deg; joints [42.781, -66.614, 72.458, -0.862, 84.079, 42.866]
  MoveL 362 to (44.16, 173.69, 0) mm, rotated rx -180 ry 0 rz -39.83 deg; joints [42.827, -66.561, 72.385, -0.862, 84.1, 42.911]
  MoveL 363 to (45.06, 174.37, 0) mm, rotated rx 180 ry 0 rz -39.83 deg; joints [42.873, -66.513, 72.318, -0.862, 84.119, 42.958]
  MoveL 364 to (46.14, 175.08, 0) mm, rotated rx 180 ry 0 rz -39.83 deg; joints [42.929, -66.463, 72.25, -0.862, 84.138, 43.013]
  MoveL 365 to (47.26, 175.73, 0) mm, rotated rx 180 ry 0 rz -39.83 deg; joints [42.986, -66.42, 72.19, -0.862, 84.156, 43.07]
  MoveL 366 to (48.42, 176.32, 0) mm, rotated rx -180 ry 0 rz -39.83 deg; joints [43.045, -66.382, 72.138, -0.862, 84.171, 43.129]
  MoveL 367 to (49.6, 176.86, 0) mm, rotated rx 180 ry 0 rz -39.83 deg; joints [43.104, -66.348, 72.092, -0.862, 84.184, 43.188]
  MoveL 368 to (51.17, 177.5, 0) mm, rotated rx 180 ry 0 rz -39.83 deg; joints [43.183, -66.309, 72.039, -0.862, 84.199, 43.266]
  MoveL 369 to (52.76, 178.08, 0) mm, rotated rx -180 ry 0 rz -39.83 deg; joints [43.262, -66.276, 71.995, -0.862, 84.211, 43.345]
  MoveL 370 to (54.37, 178.58, 0) mm, rotated rx 180 ry 0 rz -39.83 deg; joints [43.341, -66.25, 71.96, -0.862, 84.221, 43.424]
  MoveL 371 to (56.01, 178.99, 0) mm, rotated rx -180 ry 0 rz -39.83 deg; joints [43.421, -66.231, 71.934, -0.862, 84.229, 43.504]
  MoveL 372 to (57, 179.2, 0) mm, rotated rx 180 ry 0 rz -39.83 deg; joints [43.469, -66.222, 71.924, -0.862, 84.231, 43.552]
  MoveL 373 to (57.99, 179.38, 0) mm, rotated rx 180 ry 0 rz -39.83 deg; joints [43.518, -66.217, 71.917, -0.862, 84.233, 43.601]
  MoveL 374 to (58.99, 179.53, 0) mm, rotated rx -180 ry 0 rz -39.83 deg; joints [43.566, -66.214, 71.915, -0.862, 84.234, 43.649]
  MoveL 375 to (60, 179.64, 0) mm, rotated rx -180 ry 0 rz -39.83 deg; joints [43.615, -66.214, 71.916, -0.863, 84.233, 43.698]
  MoveL 376 to (61.82, 179.76, 0) mm, rotated rx 180 ry 0 rz -39.83 deg; joints [43.702, -66.222, 71.929, -0.863, 84.229, 43.785]
  MoveL 377 to (63.65, 179.75, 0) mm, rotated rx 180 ry 0 rz -39.83 deg; joints [43.788, -66.239, 71.956, -0.863, 84.221, 43.872]
  MoveL 378 to (65.46, 179.62, 0) mm, rotated rx 180 ry 0 rz -39.83 deg; joints [43.874, -66.267, 71.999, -0.863, 84.208, 43.958]
  MoveL 379 to (67.26, 179.35, 0) mm, rotated rx 180 ry 0 rz -39.83 deg; joints [43.958, -66.307, 72.057, -0.863, 84.19, 44.042]
  MoveL 380 to (68.31, 179.12, 0) mm, rotated rx -180 ry 0 rz -39.83 deg; joints [44.007, -66.337, 72.1, -0.863, 84.178, 44.091]
  MoveL 381 to (69.35, 178.85, 0) mm, rotated rx -180 ry 0 rz -39.83 deg; joints [44.055, -66.369, 72.147, -0.863, 84.164, 44.14]
  MoveL 382 to (70.39, 178.55, 0) mm, rotated rx 180 ry 0 rz -39.83 deg; joints [44.103, -66.404, 72.198, -0.863, 84.149, 44.188]
  MoveL 383 to (71.43, 178.24, 0) mm, rotated rx -180 ry 0 rz -39.83 deg; joints [44.151, -66.44, 72.249, -0.863, 84.133, 44.236]
  Establecer velocidad (1000.0 mm/s)
  MoveL 384 to (71.43, 178.24, 0) mm, rotated rx -180 ry 0 rz -39.83 deg; joints [44.151, -66.44, 72.249, -0.863, 84.133, 44.236]
  MoveL 385 to (71.43, 178.24, 20) mm, rotated rx 180 ry 0 rz -39.83 deg; joints [44.166, -66.684, 70.869, -0.861, 85.758, 44.226]
  Establecer velocidad (1000.0 mm/s)
  MoveL 386 to (33.45, 134.79, 20) mm, rotated rx -180 ry 0 rz -39.83 deg; joints [42.069, -69.999, 75.384, -0.86, 84.527, 42.147]
  MoveL 387 to (33.45, 134.79, 0) mm, rotated rx 180 ry 0 rz -39.83 deg; joints [42.054, -69.723, 76.74, -0.863, 82.895, 42.157]
  MoveL 388 to (33.45, 134.79, 0) mm, rotated rx 180 ry 0 rz -39.83 deg; joints [42.054, -69.723, 76.74, -0.863, 82.895, 42.157]
  Establecer velocidad (50.0 mm/s)
  MoveL 389 to (33.7, 134.14, 0) mm, rotated rx -180 ry 0 rz -39.83 deg; joints [42.061, -69.78, 76.818, -0.863, 82.874, 42.165]
  MoveL 390 to (33.94, 133.48, 0) mm, rotated rx -180 ry 0 rz -39.83 deg; joints [42.069, -69.838, 76.896, -0.863, 82.854, 42.172]
  MoveL 391 to (34.16, 132.82, 0) mm, rotated rx 180 ry 0 rz -39.83 deg; joints [42.075, -69.895, 76.975, -0.863, 82.833, 42.179]
  MoveL 392 to (34.36, 132.15, 0) mm, rotated rx 180 ry 0 rz -39.83 deg; joints [42.08, -69.953, 77.054, -0.863, 82.812, 42.184]
  MoveL 393 to (34.53, 131.49, 0) mm, rotated rx 180 ry 0 rz -39.83 deg; joints [42.084, -70.01, 77.131, -0.863, 82.792, 42.188]
  MoveL 394 to (34.67, 130.83, 0) mm, rotated rx 180 ry 0 rz -39.83 deg; joints [42.086, -70.067, 77.208, -0.863, 82.772, 42.19]
  MoveL 395 to (34.78, 130.16, 0) mm, rotated rx 180 ry 0 rz -39.83 deg; joints [42.086, -70.124, 77.285, -0.863, 82.752, 42.191]
  MoveL 396 to (34.86, 129.48, 0) mm, rotated rx 180 ry 0 rz -39.83 deg; joints [42.086, -70.182, 77.362, -0.863, 82.732, 42.191]
  MoveL 397 to (34.92, 128.87, 0) mm, rotated rx 180 ry 0 rz -39.83 deg; joints [42.085, -70.234, 77.433, -0.863, 82.714, 42.19]
  MoveL 398 to (34.97, 128.25, 0) mm, rotated rx 180 ry 0 rz -39.83 deg; joints [42.082, -70.286, 77.502, -0.863, 82.695, 42.188]
  MoveL 399 to (35, 127.63, 0) mm, rotated rx 180 ry 0 rz -39.83 deg; joints [42.08, -70.337, 77.572, -0.863, 82.677, 42.186]
  MoveL 400 to (35.02, 127.01, 0) mm, rotated rx 180 ry 0 rz -39.83 deg; joints [42.076, -70.389, 77.642, -0.863, 82.659, 42.183]
  MoveL 401 to (35.03, 126.2, 0) mm, rotated rx -180 ry 0 rz -39.83 deg; joints [42.071, -70.457, 77.734, -0.863, 82.636, 42.178]
  MoveL 402 to (35.04, 125.38, 0) mm, rotated rx 180 ry 0 rz -39.83 deg; joints [42.066, -70.525, 77.825, -0.863, 82.612, 42.173]
  MoveL 403 to (35.05, 124.56, 0) mm, rotated rx 180 ry 0 rz -39.83 deg; joints [42.06, -70.593, 77.916, -0.863, 82.589, 42.168]
  MoveL 404 to (35.05, 123.74, 0) mm, rotated rx 180 ry 0 rz -39.83 deg; joints [42.055, -70.661, 78.008, -0.863, 82.566, 42.163]
  MoveL 405 to (35.05, 122.71, 0) mm, rotated rx 180 ry 0 rz -39.83 deg; joints [42.048, -70.747, 78.122, -0.863, 82.537, 42.156]
  MoveL 406 to (35.05, 121.68, 0) mm, rotated rx 180 ry 0 rz -39.83 deg; joints [42.04, -70.832, 78.237, -0.863, 82.508, 42.149]
  MoveL 407 to (35.04, 120.65, 0) mm, rotated rx 180 ry 0 rz -39.83 deg; joints [42.032, -70.918, 78.351, -0.863, 82.479, 42.142]
  MoveL 408 to (35.02, 119.62, 0) mm, rotated rx 180 ry 0 rz -39.83 deg; joints [42.024, -71.003, 78.465, -0.863, 82.45, 42.134]
  MoveL 409 to (34.99, 118.86, 0) mm, rotated rx 180 ry 0 rz -39.83 deg; joints [42.017, -71.066, 78.549, -0.864, 82.429, 42.127]
  MoveL 410 to (34.95, 118.1, 0) mm, rotated rx 180 ry 0 rz -39.83 deg; joints [42.01, -71.129, 78.632, -0.864, 82.408, 42.12]
  MoveL 411 to (34.9, 117.33, 0) mm, rotated rx 180 ry 0 rz -39.83 deg; joints [42.002, -71.192, 78.716, -0.864, 82.387, 42.112]
  MoveL 412 to (34.84, 116.57, 0) mm, rotated rx 180 ry 0 rz -39.83 deg; joints [41.993, -71.254, 78.799, -0.864, 82.366, 42.104]
  MoveL 413 to (34.71, 115.28, 0) mm, rotated rx 180 ry 0 rz -39.83 deg; joints [41.978, -71.359, 78.939, -0.864, 82.331, 42.089]
  MoveL 414 to (34.56, 114, 0) mm, rotated rx -180 ry 0 rz -39.83 deg; joints [41.961, -71.464, 79.078, -0.864, 82.297, 42.072]
  MoveL 415 to (34.38, 112.71, 0) mm, rotated rx 180 ry 0 rz -39.83 deg; joints [41.942, -71.568, 79.215, -0.864, 82.263, 42.055]
  MoveL 416 to (34.18, 111.43, 0) mm, rotated rx 180 ry 0 rz -39.83 deg; joints [41.923, -71.672, 79.353, -0.864, 82.229, 42.036]
  MoveL 417 to (33.92, 109.92, 0) mm, rotated rx 180 ry 0 rz -39.83 deg; joints [41.9, -71.793, 79.513, -0.864, 82.19, 42.013]
  MoveL 418 to (33.65, 108.42, 0) mm, rotated rx 180 ry 0 rz -39.83 deg; joints [41.875, -71.914, 79.672, -0.864, 82.151, 41.989]
  MoveL 419 to (33.34, 106.93, 0) mm, rotated rx 180 ry 0 rz -39.83 deg; joints [41.848, -72.034, 79.829, -0.864, 82.113, 41.963]
  MoveL 420 to (32.99, 105.45, 0) mm, rotated rx 180 ry 0 rz -39.83 deg; joints [41.82, -72.152, 79.985, -0.864, 82.076, 41.935]
  MoveL 421 to (32.75, 104.55, 0) mm, rotated rx 180 ry 0 rz -39.83 deg; joints [41.801, -72.223, 80.078, -0.864, 82.054, 41.917]
  MoveL 422 to (32.5, 103.66, 0) mm, rotated rx 180 ry 0 rz -39.83 deg; joints [41.782, -72.294, 80.17, -0.864, 82.031, 41.898]
  MoveL 423 to (32.24, 102.78, 0) mm, rotated rx 180 ry 0 rz -39.83 deg; joints [41.762, -72.363, 80.261, -0.864, 82.01, 41.878]
  MoveL 424 to (31.95, 101.9, 0) mm, rotated rx 180 ry 0 rz -39.83 deg; joints [41.741, -72.432, 80.351, -0.864, 81.988, 41.857]
  MoveL 425 to (31.58, 100.89, 0) mm, rotated rx 180 ry 0 rz -39.83 deg; joints [41.715, -72.511, 80.454, -0.864, 81.964, 41.832]
  MoveL 426 to (31.19, 99.88, 0) mm, rotated rx 180 ry 0 rz -39.83 deg; joints [41.688, -72.589, 80.556, -0.864, 81.94, 41.805]
  MoveL 427 to (30.79, 98.88, 0) mm, rotated rx 180 ry 0 rz -39.83 deg; joints [41.66, -72.667, 80.656, -0.864, 81.916, 41.777]
  MoveL 428 to (30.37, 97.89, 0) mm, rotated rx 180 ry 0 rz -39.83 deg; joints [41.631, -72.743, 80.756, -0.864, 81.893, 41.749]
  MoveL 429 to (30.01, 97.04, 0) mm, rotated rx 180 ry 0 rz -39.83 deg; joints [41.606, -72.808, 80.841, -0.864, 81.873, 41.725]
  MoveL 430 to (29.63, 96.21, 0) mm, rotated rx 180 ry 0 rz -39.83 deg; joints [41.581, -72.873, 80.924, -0.864, 81.854, 41.699]
  MoveL 431 to (29.23, 95.39, 0) mm, rotated rx 180 ry 0 rz -39.83 deg; joints [41.554, -72.935, 81.005, -0.864, 81.835, 41.673]
  MoveL 432 to (28.79, 94.59, 0) mm, rotated rx 180 ry 0 rz -39.83 deg; joints [41.526, -72.996, 81.083, -0.864, 81.817, 41.645]
  MoveL 433 to (28.5, 94.11, 0) mm, rotated rx 180 ry 0 rz -39.83 deg; joints [41.508, -73.031, 81.129, -0.864, 81.806, 41.627]
  MoveL 434 to (28.2, 93.65, 0) mm, rotated rx -180 ry 0 rz -39.83 deg; joints [41.489, -73.065, 81.173, -0.864, 81.796, 41.608]
  MoveL 435 to (27.88, 93.19, 0) mm, rotated rx 180 ry 0 rz -39.83 deg; joints [41.469, -73.099, 81.216, -0.864, 81.786, 41.588]
  MoveL 436 to (27.54, 92.74, 0) mm, rotated rx 180 ry 0 rz -39.83 deg; joints [41.448, -73.132, 81.258, -0.864, 81.776, 41.568]
  MoveL 437 to (27.25, 92.38, 0) mm, rotated rx 180 ry 0 rz -39.83 deg; joints [41.431, -73.158, 81.292, -0.864, 81.769, 41.55]
  MoveL 438 to (26.95, 92.03, 0) mm, rotated rx 180 ry 0 rz -39.83 deg; joints [41.412, -73.183, 81.325, -0.864, 81.761, 41.532]
  MoveL 439 to (26.62, 91.7, 0) mm, rotated rx 180 ry 0 rz -39.83 deg; joints [41.393, -73.206, 81.354, -0.864, 81.755, 41.513]
  MoveL 440 to (26.26, 91.41, 0) mm, rotated rx 180 ry 0 rz -39.83 deg; joints [41.373, -73.226, 81.379, -0.864, 81.749, 41.493]
  MoveL 441 to (25.97, 91.21, 0) mm, rotated rx 180 ry 0 rz -39.83 deg; joints [41.357, -73.238, 81.394, -0.864, 81.745, 41.477]
  MoveL 442 to (25.67, 91.04, 0) mm, rotated rx -180 ry 0 rz -39.83 deg; joints [41.34, -73.248, 81.407, -0.864, 81.742, 41.46]
  MoveL 443 to (25.36, 90.88, 0) mm, rotated rx 180 ry 0 rz -39.83 deg; joints [41.323, -73.258, 81.419, -0.864, 81.74, 41.443]
  MoveL 444 to (25.04, 90.72, 0) mm, rotated rx 180 ry 0 rz -39.83 deg; joints [41.305, -73.266, 81.43, -0.864, 81.737, 41.426]
  MoveL 445 to (24.83, 90.62, 0) mm, rotated rx 180 ry 0 rz -39.83 deg; joints [41.294, -73.272, 81.437, -0.864, 81.736, 41.414]
  MoveL 446 to (24.61, 90.52, 0) mm, rotated rx -180 ry 0 rz -39.83 deg; joints [41.282, -73.278, 81.444, -0.864, 81.734, 41.402]
  MoveL 447 to (24.38, 90.43, 0) mm, rotated rx 180 ry 0 rz -39.83 deg; joints [41.27, -73.282, 81.449, -0.864, 81.733, 41.39]
  MoveL 448 to (24.15, 90.37, 0) mm, rotated rx 180 ry 0 rz -39.83 deg; joints [41.257, -73.284, 81.452, -0.864, 81.732, 41.378]
  MoveL 449 to (24, 90.34, 0) mm, rotated rx 180 ry 0 rz -39.83 deg; joints [41.249, -73.285, 81.452, -0.864, 81.732, 41.37]
  MoveL 450 to (23.85, 90.33, 0) mm, rotated rx 180 ry 0 rz -39.83 deg; joints [41.242, -73.284, 81.451, -0.864, 81.733, 41.362]
  MoveL 451 to (23.7, 90.34, 0) mm, rotated rx -180 ry 0 rz -39.83 deg; joints [41.234, -73.281, 81.447, -0.864, 81.734, 41.354]
  MoveL 452 to (23.56, 90.37, 0) mm, rotated rx 180 ry 0 rz -39.83 deg; joints [41.227, -73.277, 81.442, -0.864, 81.735, 41.347]
  MoveL 453 to (23.49, 90.39, 0) mm, rotated rx 180 ry 0 rz -39.83 deg; joints [41.224, -73.274, 81.438, -0.864, 81.736, 41.344]
  MoveL 454 to (23.42, 90.42, 0) mm, rotated rx -180 ry 0 rz -39.83 deg; joints [41.221, -73.271, 81.434, -0.864, 81.737, 41.341]
  MoveL 455 to (23.35, 90.45, 0) mm, rotated rx 180 ry 0 rz -39.83 deg; joints [41.217, -73.267, 81.429, -0.864, 81.738, 41.338]
  MoveL 456 to (23.29, 90.49, 0) mm, rotated rx 180 ry 0 rz -39.83 deg; joints [41.214, -73.264, 81.424, -0.864, 81.739, 41.335]
  MoveL 457 to (23.2, 90.54, 0) mm, rotated rx 180 ry 0 rz -39.83 deg; joints [41.21, -73.259, 81.417, -0.864, 81.741, 41.33]
  MoveL 458 to (23.11, 90.59, 0) mm, rotated rx 180 ry 0 rz -39.83 deg; joints [41.206, -73.253, 81.41, -0.864, 81.742, 41.326]
  MoveL 459 to (23.02, 90.64, 0) mm, rotated rx 180 ry 0 rz -39.83 deg; joints [41.202, -73.248, 81.403, -0.864, 81.744, 41.322]
  MoveL 460 to (22.93, 90.69, 0) mm, rotated rx 180 ry 0 rz -39.83 deg; joints [41.198, -73.242, 81.396, -0.864, 81.746, 41.318]
  MoveL 461 to (22.75, 90.83, 0) mm, rotated rx -180 ry 0 rz -39.83 deg; joints [41.19, -73.228, 81.378, -0.864, 81.75, 41.31]
  MoveL 462 to (22.57, 90.99, 0) mm, rotated rx 180 ry 0 rz -39.83 deg; joints [41.182, -73.214, 81.358, -0.864, 81.754, 41.302]
  MoveL 463 to (22.41, 91.15, 0) mm, rotated rx -180 ry 0 rz -39.83 deg; joints [41.175, -73.198, 81.338, -0.863, 81.759, 41.295]
  MoveL 464 to (22.25, 91.32, 0) mm, rotated rx 180 ry 0 rz -39.83 deg; joints [41.168, -73.182, 81.317, -0.863, 81.764, 41.288]
  MoveL 465 to (21.92, 91.67, 0) mm, rotated rx 180 ry 0 rz -39.83 deg; joints [41.154, -73.149, 81.274, -0.863, 81.774, 41.274]
  MoveL 466 to (21.59, 92.02, 0) mm, rotated rx 180 ry 0 rz -39.83 deg; joints [41.141, -73.116, 81.23, -0.863, 81.784, 41.26]
  MoveL 467 to (21.28, 92.38, 0) mm, rotated rx 180 ry 0 rz -39.83 deg; joints [41.127, -73.083, 81.186, -0.863, 81.794, 41.247]
  MoveL 468 to (20.97, 92.74, 0) mm, rotated rx -180 ry 0 rz -39.83 deg; joints [41.115, -73.049, 81.142, -0.863, 81.805, 41.234]
  MoveL 469 to (20.65, 93.14, 0) mm, rotated rx -180 ry 0 rz -39.83 deg; joints [41.102, -73.012, 81.094, -0.863, 81.816, 41.221]
  MoveL 470 to (20.35, 93.55, 0) mm, rotated rx -180 ry 0 rz -39.83 deg; joints [41.09, -72.974, 81.044, -0.863, 81.828, 41.209]
  MoveL 471 to (20.05, 93.97, 0) mm, rotated rx -180 ry 0 rz -39.83 deg; joints [41.078, -72.937, 80.995, -0.863, 81.839, 41.197]
  MoveL 472 to (19.75, 94.38, 0) mm, rotated rx 180 ry 0 rz -39.83 deg; joints [41.066, -72.899, 80.945, -0.863, 81.851, 41.185]
  MoveL 473 to (19.49, 94.74, 0) mm, rotated rx -180 ry 0 rz -39.83 deg; joints [41.056, -72.866, 80.902, -0.863, 81.861, 41.174]
  MoveL 474 to (19.23, 95.1, 0) mm, rotated rx -180 ry 0 rz -39.83 deg; joints [41.046, -72.833, 80.859, -0.863, 81.871, 41.164]
  MoveL 475 to (18.98, 95.46, 0) mm, rotated rx 180 ry 0 rz -39.83 deg; joints [41.036, -72.8, 80.815, -0.863, 81.882, 41.154]
  MoveL 476 to (18.74, 95.84, 0) mm, rotated rx 180 ry 0 rz -39.83 deg; joints [41.027, -72.766, 80.771, -0.863, 81.892, 41.145]
  MoveL 477 to (18.61, 96.05, 0) mm, rotated rx 180 ry 0 rz -39.83 deg; joints [41.022, -72.746, 80.745, -0.863, 81.898, 41.14]
  MoveL 478 to (18.48, 96.27, 0) mm, rotated rx -180 ry 0 rz -39.83 deg; joints [41.018, -72.727, 80.719, -0.863, 81.904, 41.135]
  MoveL 479 to (18.36, 96.5, 0) mm, rotated rx 180 ry 0 rz -39.83 deg; joints [41.013, -72.707, 80.693, -0.863, 81.911, 41.131]
  MoveL 480 to (18.24, 96.72, 0) mm, rotated rx 180 ry 0 rz -39.83 deg; joints [41.009, -72.687, 80.667, -0.863, 81.917, 41.126]
  Establecer velocidad (1000.0 mm/s)
  MoveL 481 to (18.24, 96.72, 0) mm, rotated rx 180 ry 0 rz -39.83 deg; joints [41.009, -72.687, 80.667, -0.863, 81.917, 41.126]
  MoveL 482 to (18.24, 96.72, 20) mm, rotated rx 180 ry 0 rz -39.83 deg; joints [41.024, -72.989, 79.326, -0.86, 83.56, 41.117]
  Establecer velocidad (1000.0 mm/s)
  MoveL 483 to (33.45, 134.79, 20) mm, rotated rx -180 ry 0 rz -39.83 deg; joints [42.069, -69.999, 75.384, -0.86, 84.527, 42.147]
  MoveL 484 to (33.45, 134.79, 0) mm, rotated rx 180 ry 0 rz -39.83 deg; joints [42.054, -69.723, 76.74, -0.863, 82.895, 42.157]
  MoveL 485 to (33.45, 134.79, 0) mm, rotated rx 180 ry 0 rz -39.83 deg; joints [42.054, -69.723, 76.74, -0.863, 82.895, 42.157]
  Establecer velocidad (50.0 mm/s)
  MoveL 486 to (33.28, 135.18, 0) mm, rotated rx 180 ry 0 rz -39.83 deg; joints [42.048, -69.688, 76.693, -0.863, 82.907, 42.151]
  MoveL 487 to (33.1, 135.56, 0) mm, rotated rx 180 ry 0 rz -39.83 deg; joints [42.042, -69.654, 76.646, -0.863, 82.92, 42.144]
  MoveL 488 to (32.91, 135.94, 0) mm, rotated rx 180 ry 0 rz -39.83 deg; joints [42.035, -69.621, 76.601, -0.863, 82.932, 42.137]
  MoveL 489 to (32.69, 136.3, 0) mm, rotated rx 180 ry 0 rz -39.83 deg; joints [42.027, -69.588, 76.556, -0.863, 82.944, 42.129]
  MoveL 490 to (32.47, 136.61, 0) mm, rotated rx 180 ry 0 rz -39.83 deg; joints [42.018, -69.559, 76.516, -0.862, 82.954, 42.12]
  MoveL 491 to (32.22, 136.91, 0) mm, rotated rx 180 ry 0 rz -39.83 deg; joints [42.008, -69.531, 76.478, -0.862, 82.964, 42.11]
  MoveL 492 to (31.96, 137.2, 0) mm, rotated rx 180 ry 0 rz -39.83 deg; joints [41.997, -69.504, 76.441, -0.862, 82.974, 42.099]
  MoveL 493 to (31.67, 137.46, 0) mm, rotated rx 180 ry 0 rz -39.83 deg; joints [41.985, -69.479, 76.407, -0.862, 82.983, 42.087]
  MoveL 494 to (31.47, 137.62, 0) mm, rotated rx 180 ry 0 rz -39.83 deg; joints [41.976, -69.463, 76.385, -0.862, 82.989, 42.078]
  MoveL 495 to (31.25, 137.76, 0) mm, rotated rx 180 ry 0 rz -39.83 deg; joints [41.967, -69.448, 76.364, -0.862, 82.995, 42.068]
  MoveL 496 to (31.03, 137.89, 0) mm, rotated rx 180 ry 0 rz -39.83 deg; joints [41.957, -69.435, 76.346, -0.862, 83, 42.058]
  MoveL 497 to (30.79, 137.99, 0) mm, rotated rx 180 ry 0 rz -39.83 deg; joints [41.946, -69.424, 76.331, -0.862, 83.004, 42.047]
  MoveL 498 to (30.56, 138.06, 0) mm, rotated rx 180 ry 0 rz -39.83 deg; joints [41.935, -69.416, 76.319, -0.862, 83.007, 42.036]
  MoveL 499 to (30.32, 138.1, 0) mm, rotated rx 180 ry 0 rz -39.83 deg; joints [41.924, -69.41, 76.31, -0.862, 83.009, 42.025]
  MoveL 500 to (30.08, 138.11, 0) mm, rotated rx -180 ry 0 rz -39.83 deg; joints [41.912, -69.406, 76.305, -0.862, 83.011, 42.013]
  MoveL 501 to (29.84, 138.09, 0) mm, rotated rx 180 ry 0 rz -39.83 deg; joints [41.9, -69.404, 76.302, -0.862, 83.012, 42.001]
  MoveL 502 to (29.65, 138.06, 0) mm, rotated rx 180 ry 0 rz -39.83 deg; joints [41.891, -69.404, 76.302, -0.862, 83.012, 41.992]
  MoveL 503 to (29.47, 138.02, 0) mm, rotated rx 180 ry 0 rz -39.83 deg; joints [41.882, -69.406, 76.304, -0.862, 83.011, 41.983]
  MoveL 504 to (29.29, 137.97, 0) mm, rotated rx 180 ry 0 rz -39.83 deg; joints [41.872, -69.408, 76.307, -0.862, 83.01, 41.973]
  MoveL 505 to (29.11, 137.91, 0) mm, rotated rx 180 ry 0 rz -39.83 deg; joints [41.863, -69.411, 76.31, -0.862, 83.01, 41.964]
  MoveL 506 to (29.11, 137.91, 0) mm, rotated rx 180 ry 0 rz -39.83 deg; joints [41.863, -69.411, 76.31, -0.862, 83.01, 41.964]
  MoveL 507 to (28, 137.2, 0) mm, rotated rx 180 ry 0 rz -39.83 deg; joints [41.804, -69.456, 76.371, -0.862, 82.994, 41.905]
  MoveL 508 to (26.89, 136.49, 0) mm, rotated rx 180 ry 0 rz -39.83 deg; joints [41.745, -69.503, 76.433, -0.862, 82.977, 41.846]
  MoveL 509 to (25.8, 135.74, 0) mm, rotated rx -180 ry 0 rz -39.83 deg; joints [41.686, -69.552, 76.498, -0.862, 82.96, 41.788]
  MoveL 510 to (24.74, 134.96, 0) mm, rotated rx 180 ry 0 rz -39.83 deg; joints [41.628, -69.604, 76.567, -0.862, 82.942, 41.73]
  MoveL 511 to (23.05, 133.56, 0) mm, rotated rx 180 ry 0 rz -39.83 deg; joints [41.535, -69.7, 76.695, -0.862, 82.909, 41.637]
  MoveL 512 to (21.47, 132.02, 0) mm, rotated rx 180 ry 0 rz -39.83 deg; joints [41.446, -69.808, 76.84, -0.862, 82.871, 41.549]
  MoveL 513 to (20.03, 130.36, 0) mm, rotated rx 180 ry 0 rz -39.83 deg; joints [41.363, -69.929, 77.001, -0.862, 82.829, 41.467]
  MoveL 514 to (18.76, 128.58, 0) mm, rotated rx 180 ry 0 rz -39.83 deg; joints [41.287, -70.061, 77.178, -0.862, 82.783, 41.391]
  MoveL 515 to (17.96, 127.24, 0) mm, rotated rx -180 ry 0 rz -39.83 deg; joints [41.238, -70.161, 77.313, -0.862, 82.748, 41.342]
  MoveL 516 to (17.24, 125.86, 0) mm, rotated rx -180 ry 0 rz -39.83 deg; joints [41.192, -70.267, 77.454, -0.862, 82.712, 41.297]
  MoveL 517 to (16.59, 124.45, 0) mm, rotated rx 180 ry 0 rz -39.83 deg; joints [41.148, -70.376, 77.6, -0.862, 82.674, 41.254]
  MoveL 518 to (15.97, 123.01, 0) mm, rotated rx 180 ry 0 rz -39.83 deg; joints [41.107, -70.487, 77.749, -0.862, 82.636, 41.213]
  MoveL 519 to (15.43, 121.67, 0) mm, rotated rx 180 ry 0 rz -39.83 deg; joints [41.069, -70.591, 77.888, -0.862, 82.601, 41.176]
  MoveL 520 to (14.94, 120.31, 0) mm, rotated rx 180 ry 0 rz -39.83 deg; joints [41.034, -70.698, 78.03, -0.862, 82.565, 41.142]
  MoveL 521 to (14.51, 118.94, 0) mm, rotated rx 180 ry 0 rz -39.83 deg; joints [41.002, -70.806, 78.174, -0.862, 82.528, 41.11]
  MoveL 522 to (14.18, 117.54, 0) mm, rotated rx -180 ry 0 rz -39.83 deg; joints [40.974, -70.917, 78.322, -0.862, 82.491, 41.083]
  MoveL 523 to (13.91, 115.68, 0) mm, rotated rx 180 ry 0 rz -39.83 deg; joints [40.946, -71.067, 78.523, -0.862, 82.44, 41.055]
  MoveL 524 to (13.8, 113.79, 0) mm, rotated rx 180 ry 0 rz -39.83 deg; joints [40.925, -71.222, 78.729, -0.862, 82.388, 41.036]
  MoveL 525 to (13.82, 111.89, 0) mm, rotated rx -180 ry 0 rz -39.83 deg; joints [40.911, -71.379, 78.938, -0.862, 82.336, 41.022]
  MoveL 526 to (13.94, 109.99, 0) mm, rotated rx 180 ry 0 rz -39.83 deg; joints [40.902, -71.537, 79.148, -0.862, 82.284, 41.013]
  MoveL 527 to (14.05, 108.82, 0) mm, rotated rx 180 ry 0 rz -39.83 deg; joints [40.898, -71.636, 79.278, -0.862, 82.252, 41.01]
  MoveL 528 to (14.19, 107.66, 0) mm, rotated rx 180 ry 0 rz -39.83 deg; joints [40.895, -71.734, 79.408, -0.862, 82.22, 41.008]
  MoveL 529 to (14.37, 106.5, 0) mm, rotated rx -180 ry 0 rz -39.83 deg; joints [40.895, -71.831, 79.537, -0.862, 82.189, 41.008]
  MoveL 530 to (14.6, 105.35, 0) mm, rotated rx 180 ry 0 rz -39.83 deg; joints [40.897, -71.929, 79.667, -0.862, 82.157, 41.01]
  MoveL 531 to (14.91, 104.08, 0) mm, rotated rx 180 ry 0 rz -39.83 deg; joints [40.902, -72.038, 79.81, -0.862, 82.122, 41.016]
  MoveL 532 to (15.29, 102.83, 0) mm, rotated rx 180 ry 0 rz -39.83 deg; joints [40.911, -72.146, 79.953, -0.862, 82.087, 41.026]
  MoveL 533 to (15.74, 101.6, 0) mm, rotated rx 180 ry 0 rz -39.83 deg; joints [40.923, -72.253, 80.095, -0.862, 82.053, 41.038]
  MoveL 534 to (16.25, 100.4, 0) mm, rotated rx -180 ry 0 rz -39.83 deg; joints [40.939, -72.358, 80.234, -0.862, 82.02, 41.055]
  MoveL 535 to (16.71, 99.46, 0) mm, rotated rx 180 ry 0 rz -39.83 deg; joints [40.955, -72.442, 80.344, -0.863, 81.994, 41.071]
  MoveL 536 to (17.2, 98.54, 0) mm, rotated rx 180 ry 0 rz -39.83 deg; joints [40.972, -72.524, 80.452, -0.863, 81.968, 41.088]
  MoveL 537 to (17.71, 97.63, 0) mm, rotated rx 180 ry 0 rz -39.83 deg; joints [40.99, -72.606, 80.56, -0.863, 81.942, 41.107]
  MoveL 538 to (18.24, 96.72, 0) mm, rotated rx 180 ry 0 rz -39.83 deg; joints [41.009, -72.687, 80.667, -0.863, 81.917, 41.126]
  Establecer velocidad (1000.0 mm/s)
  MoveL 539 to (18.24, 96.72, 0) mm, rotated rx 180 ry 0 rz -39.83 deg; joints [41.009, -72.687, 80.667, -0.863, 81.917, 41.126]
  MoveL 540 to (18.24, 96.72, 20) mm, rotated rx 180 ry 0 rz -39.83 deg; joints [41.024, -72.989, 79.326, -0.86, 83.56, 41.117]
  Establecer velocidad (1000.0 mm/s)
  MoveL 541 to (34.98, 89.11, 20) mm, rotated rx 180 ry 0 rz -39.83 deg; joints [41.815, -73.829, 80.433, -0.862, 83.304, 41.911]
  MoveL 542 to (34.98, 89.11, 0) mm, rotated rx -180 ry 0 rz -39.83 deg; joints [41.799, -73.52, 81.771, -0.865, 81.657, 41.921]
  MoveL 543 to (34.98, 89.11, 0) mm, rotated rx -180 ry 0 rz -39.83 deg; joints [41.799, -73.52, 81.771, -0.865, 81.657, 41.921]
  Establecer velocidad (50.0 mm/s)
  MoveL 544 to (35.52, 89.26, 0) mm, rotated rx 180 ry 0 rz -39.83 deg; joints [41.828, -73.514, 81.765, -0.865, 81.658, 41.949]
  MoveL 545 to (36.06, 89.39, 0) mm, rotated rx 180 ry 0 rz -39.83 deg; joints [41.856, -73.51, 81.759, -0.865, 81.659, 41.977]
  MoveL 546 to (36.59, 89.51, 0) mm, rotated rx 180 ry 0 rz -39.83 deg; joints [41.884, -73.506, 81.755, -0.865, 81.66, 42.006]
  MoveL 547 to (37.14, 89.61, 0) mm, rotated rx -180 ry 0 rz -39.83 deg; joints [41.913, -73.504, 81.754, -0.865, 81.66, 42.034]
  MoveL 548 to (38.25, 89.71, 0) mm, rotated rx -180 ry 0 rz -39.83 deg; joints [41.97, -73.509, 81.762, -0.865, 81.658, 42.092]
  MoveL 549 to (39.38, 89.69, 0) mm, rotated rx 180 ry 0 rz -39.83 deg; joints [42.028, -73.524, 81.782, -0.865, 81.653, 42.149]
  MoveL 550 to (40.5, 89.57, 0) mm, rotated rx 180 ry 0 rz -39.83 deg; joints [42.084, -73.547, 81.813, -0.865, 81.646, 42.206]
  MoveL 551 to (41.61, 89.36, 0) mm, rotated rx 180 ry 0 rz -39.83 deg; joints [42.139, -73.576, 81.853, -0.865, 81.637, 42.261]
  MoveL 552 to (42.52, 89.13, 0) mm, rotated rx 180 ry 0 rz -39.83 deg; joints [42.184, -73.606, 81.892, -0.865, 81.628, 42.306]
  MoveL 553 to (43.42, 88.85, 0) mm, rotated rx 180 ry 0 rz -39.83 deg; joints [42.228, -73.638, 81.935, -0.866, 81.618, 42.35]
  MoveL 554 to (44.3, 88.54, 0) mm, rotated rx -180 ry 0 rz -39.83 deg; joints [42.271, -73.674, 81.982, -0.866, 81.607, 42.394]
  MoveL 555 to (45.17, 88.2, 0) mm, rotated rx 180 ry 0 rz -39.83 deg; joints [42.313, -73.712, 82.032, -0.866, 81.596, 42.436]
  MoveL 556 to (45.87, 87.91, 0) mm, rotated rx 180 ry 0 rz -39.83 deg; joints [42.347, -73.743, 82.074, -0.866, 81.586, 42.47]
  MoveL 557 to (46.55, 87.61, 0) mm, rotated rx -180 ry 0 rz -39.83 deg; joints [42.38, -73.776, 82.117, -0.866, 81.576, 42.503]
  MoveL 558 to (47.23, 87.29, 0) mm, rotated rx 180 ry 0 rz -39.83 deg; joints [42.412, -73.809, 82.161, -0.866, 81.566, 42.536]
  MoveL 559 to (47.91, 86.96, 0) mm, rotated rx -180 ry 0 rz -39.83 deg; joints [42.445, -73.844, 82.206, -0.866, 81.556, 42.568]
  MoveL 560 to (48.69, 86.56, 0) mm, rotated rx 180 ry 0 rz -39.83 deg; joints [42.482, -73.885, 82.26, -0.866, 81.543, 42.606]
  MoveL 561 to (49.47, 86.14, 0) mm, rotated rx 180 ry 0 rz -39.83 deg; joints [42.519, -73.928, 82.317, -0.866, 81.531, 42.643]
  MoveL 562 to (50.23, 85.69, 0) mm, rotated rx 180 ry 0 rz -39.83 deg; joints [42.555, -73.973, 82.375, -0.866, 81.517, 42.679]
  MoveL 563 to (50.97, 85.22, 0) mm, rotated rx 180 ry 0 rz -39.83 deg; joints [42.59, -74.02, 82.436, -0.866, 81.504, 42.714]
  MoveL 564 to (51.75, 84.68, 0) mm, rotated rx -180 ry 0 rz -39.83 deg; joints [42.626, -74.072, 82.504, -0.866, 81.488, 42.751]
  MoveL 565 to (52.51, 84.12, 0) mm, rotated rx -180 ry 0 rz -39.83 deg; joints [42.661, -74.127, 82.575, -0.867, 81.472, 42.786]
  MoveL 566 to (53.24, 83.52, 0) mm, rotated rx 180 ry 0 rz -39.83 deg; joints [42.695, -74.183, 82.649, -0.867, 81.456, 42.82]
  MoveL 567 to (53.96, 82.9, 0) mm, rotated rx 180 ry 0 rz -39.83 deg; joints [42.728, -74.242, 82.724, -0.867, 81.439, 42.853]
  MoveL 568 to (54.58, 82.34, 0) mm, rotated rx 180 ry 0 rz -39.83 deg; joints [42.756, -74.294, 82.792, -0.867, 81.424, 42.881]
  MoveL 569 to (55.18, 81.77, 0) mm, rotated rx 180 ry 0 rz -39.83 deg; joints [42.783, -74.347, 82.862, -0.867, 81.409, 42.909]
  MoveL 570 to (55.78, 81.18, 0) mm, rotated rx 180 ry 0 rz -39.83 deg; joints [42.81, -74.402, 82.932, -0.867, 81.393, 42.936]
  MoveL 571 to (56.36, 80.59, 0) mm, rotated rx 180 ry 0 rz -39.83 deg; joints [42.836, -74.457, 83.003, -0.867, 81.378, 42.962]
  MoveL 572 to (56.95, 79.96, 0) mm, rotated rx 180 ry 0 rz -39.83 deg; joints [42.863, -74.515, 83.077, -0.867, 81.361, 42.989]
  MoveL 573 to (57.54, 79.32, 0) mm, rotated rx 180 ry 0 rz -39.83 deg; joints [42.889, -74.573, 83.152, -0.867, 81.345, 43.015]
  MoveL 574 to (58.11, 78.67, 0) mm, rotated rx 180 ry 0 rz -39.83 deg; joints [42.914, -74.632, 83.228, -0.867, 81.329, 43.041]
  MoveL 575 to (58.68, 78.02, 0) mm, rotated rx 180 ry 0 rz -39.83 deg; joints [42.939, -74.691, 83.305, -0.867, 81.312, 43.067]
  MoveL 576 to (59.22, 77.38, 0) mm, rotated rx -180 ry 0 rz -39.83 deg; joints [42.963, -74.749, 83.379, -0.867, 81.296, 43.091]
  MoveL 577 to (59.76, 76.74, 0) mm, rotated rx 180 ry 0 rz -39.83 deg; joints [42.987, -74.807, 83.453, -0.867, 81.28, 43.115]
  MoveL 578 to (60.3, 76.1, 0) mm, rotated rx 180 ry 0 rz -39.83 deg; joints [43.011, -74.865, 83.528, -0.867, 81.264, 43.139]
  MoveL 579 to (60.83, 75.45, 0) mm, rotated rx 180 ry 0 rz -39.83 deg; joints [43.034, -74.923, 83.603, -0.868, 81.248, 43.163]
  MoveL 580 to (61.35, 74.83, 0) mm, rotated rx 180 ry 0 rz -39.83 deg; joints [43.057, -74.98, 83.675, -0.868, 81.232, 43.186]
  MoveL 581 to (61.86, 74.2, 0) mm, rotated rx 180 ry 0 rz -39.83 deg; joints [43.08, -75.037, 83.748, -0.868, 81.217, 43.209]
  MoveL 582 to (62.36, 73.55, 0) mm, rotated rx 180 ry 0 rz -39.83 deg; joints [43.101, -75.095, 83.821, -0.868, 81.201, 43.23]
  MoveL 583 to (62.82, 72.89, 0) mm, rotated rx 180 ry 0 rz -39.83 deg; joints [43.121, -75.154, 83.897, -0.868, 81.185, 43.25]
  MoveL 584 to (63.26, 72.18, 0) mm, rotated rx -180 ry 0 rz -39.83 deg; joints [43.14, -75.216, 83.976, -0.868, 81.168, 43.269]
  MoveL 585 to (63.68, 71.46, 0) mm, rotated rx -180 ry 0 rz -39.83 deg; joints [43.157, -75.279, 84.057, -0.868, 81.151, 43.286]
  MoveL 586 to (64.08, 70.72, 0) mm, rotated rx 180 ry 0 rz -39.83 deg; joints [43.173, -75.343, 84.138, -0.868, 81.134, 43.303]
  MoveL 587 to (64.48, 69.99, 0) mm, rotated rx 180 ry 0 rz -39.83 deg; joints [43.189, -75.408, 84.219, -0.868, 81.117, 43.319]
  MoveL 588 to (64.96, 69.15, 0) mm, rotated rx 180 ry 0 rz -39.83 deg; joints [43.209, -75.482, 84.313, -0.868, 81.098, 43.339]
  MoveL 589 to (65.45, 68.3, 0) mm, rotated rx 180 ry 0 rz -39.83 deg; joints [43.229, -75.555, 84.407, -0.868, 81.078, 43.36]
  MoveL 590 to (65.93, 67.46, 0) mm, rotated rx 180 ry 0 rz -39.83 deg; joints [43.249, -75.629, 84.5, -0.868, 81.059, 43.38]
  MoveL 591 to (66.38, 66.6, 0) mm, rotated rx 180 ry 0 rz -39.83 deg; joints [43.267, -75.704, 84.595, -0.868, 81.039, 43.399]
  MoveL 592 to (66.71, 65.93, 0) mm, rotated rx 180 ry 0 rz -39.83 deg; joints [43.28, -75.762, 84.668, -0.868, 81.025, 43.412]
  MoveL 593 to (67.01, 65.25, 0) mm, rotated rx -180 ry 0 rz -39.83 deg; joints [43.291, -75.821, 84.742, -0.868, 81.009, 43.423]
  MoveL 594 to (67.29, 64.56, 0) mm, rotated rx -180 ry 0 rz -39.83 deg; joints [43.301, -75.88, 84.816, -0.868, 80.994, 43.434]
  MoveL 595 to (67.54, 63.87, 0) mm, rotated rx 180 ry 0 rz -39.83 deg; joints [43.311, -75.939, 84.891, -0.869, 80.979, 43.443]
  MoveL 596 to (67.82, 63.05, 0) mm, rotated rx 180 ry 0 rz -39.83 deg; joints [43.32, -76.009, 84.979, -0.869, 80.961, 43.453]
  MoveL 597 to (68.08, 62.22, 0) mm, rotated rx 180 ry 0 rz -39.83 deg; joints [43.329, -76.079, 85.066, -0.869, 80.944, 43.462]
  MoveL 598 to (68.32, 61.39, 0) mm, rotated rx 180 ry 0 rz -39.83 deg; joints [43.336, -76.149, 85.154, -0.869, 80.926, 43.469]
  MoveL 599 to (68.54, 60.55, 0) mm, rotated rx 180 ry 0 rz -39.83 deg; joints [43.342, -76.22, 85.243, -0.869, 80.909, 43.476]
  MoveL 600 to (68.79, 59.49, 0) mm, rotated rx 180 ry 0 rz -39.83 deg; joints [43.349, -76.31, 85.355, -0.869, 80.886, 43.483]
  MoveL 601 to (69.02, 58.42, 0) mm, rotated rx -180 ry 0 rz -39.83 deg; joints [43.354, -76.4, 85.467, -0.869, 80.864, 43.488]
  MoveL 602 to (69.21, 57.34, 0) mm, rotated rx 180 ry 0 rz -39.83 deg; joints [43.357, -76.49, 85.579, -0.869, 80.842, 43.492]
  MoveL 603 to (69.37, 56.25, 0) mm, rotated rx -180 ry 0 rz -39.83 deg; joints [43.359, -76.58, 85.692, -0.869, 80.82, 43.494]
  MoveL 604 to (69.45, 55.53, 0) mm, rotated rx 180 ry 0 rz -39.83 deg; joints [43.358, -76.64, 85.766, -0.869, 80.806, 43.493]
  MoveL 605 to (69.5, 54.8, 0) mm, rotated rx -180 ry 0 rz -39.83 deg; joints [43.357, -76.7, 85.84, -0.869, 80.791, 43.492]
  MoveL 606 to (69.53, 54.08, 0) mm, rotated rx -180 ry 0 rz -39.83 deg; joints [43.354, -76.759, 85.914, -0.869, 80.777, 43.489]
  MoveL 607 to (69.53, 53.35, 0) mm, rotated rx 180 ry 0 rz -39.83 deg; joints [43.349, -76.819, 85.987, -0.869, 80.763, 43.485]
  MoveL 608 to (69.5, 52.63, 0) mm, rotated rx 180 ry 0 rz -39.83 deg; joints [43.343, -76.878, 86.06, -0.869, 80.749, 43.479]
  MoveL 609 to (69.43, 51.9, 0) mm, rotated rx 180 ry 0 rz -39.83 deg; joints [43.335, -76.937, 86.133, -0.869, 80.735, 43.471]
  MoveL 610 to (69.33, 51.18, 0) mm, rotated rx -180 ry 0 rz -39.83 deg; joints [43.325, -76.995, 86.204, -0.869, 80.722, 43.461]
  MoveL 611 to (69.2, 50.46, 0) mm, rotated rx 180 ry 0 rz -39.83 deg; joints [43.313, -77.052, 86.275, -0.869, 80.708, 43.45]
  MoveL 612 to (69.05, 49.79, 0) mm, rotated rx -180 ry 0 rz -39.83 deg; joints [43.301, -77.105, 86.34, -0.869, 80.696, 43.437]
  MoveL 613 to (68.87, 49.14, 0) mm, rotated rx 180 ry 0 rz -39.83 deg; joints [43.287, -77.157, 86.403, -0.869, 80.684, 43.424]
  MoveL 614 to (68.64, 48.51, 0) mm, rotated rx 180 ry 0 rz -39.83 deg; joints [43.271, -77.207, 86.464, -0.869, 80.673, 43.408]
  MoveL 615 to (68.37, 47.89, 0) mm, rotated rx 180 ry 0 rz -39.83 deg; joints [43.252, -77.254, 86.522, -0.869, 80.662, 43.39]
  MoveL 616 to (68, 47.2, 0) mm, rotated rx 180 ry 0 rz -39.83 deg; joints [43.228, -77.307, 86.586, -0.869, 80.65, 43.365]
  MoveL 617 to (67.56, 46.55, 0) mm, rotated rx 180 ry 0 rz -39.83 deg; joints [43.2, -77.356, 86.646, -0.869, 80.639, 43.338]
  MoveL 618 to (67.08, 45.92, 0) mm, rotated rx 180 ry 0 rz -39.83 deg; joints [43.17, -77.402, 86.702, -0.869, 80.629, 43.308]
  MoveL 619 to (66.55, 45.32, 0) mm, rotated rx -180 ry 0 rz -39.83 deg; joints [43.138, -77.446, 86.756, -0.869, 80.619, 43.276]
  MoveL 620 to (65.96, 44.72, 0) mm, rotated rx 180 ry 0 rz -39.83 deg; joints [43.102, -77.49, 86.808, -0.869, 80.61, 43.24]
  MoveL 621 to (65.32, 44.17, 0) mm, rotated rx 180 ry 0 rz -39.83 deg; joints [43.065, -77.529, 86.855, -0.869, 80.601, 43.203]
  MoveL 622 to (64.63, 43.7, 0) mm, rotated rx 180 ry 0 rz -39.83 deg; joints [43.025, -77.56, 86.892, -0.869, 80.595, 43.163]
  MoveL 623 to (63.9, 43.34, 0) mm, rotated rx 180 ry 0 rz -39.83 deg; joints [42.983, -77.582, 86.918, -0.869, 80.59, 43.121]
  MoveL 624 to (63.23, 43.13, 0) mm, rotated rx 180 ry 0 rz -39.83 deg; joints [42.946, -77.592, 86.93, -0.869, 80.588, 43.084]
  MoveL 625 to (62.52, 43.01, 0) mm, rotated rx -180 ry 0 rz -39.83 deg; joints [42.907, -77.595, 86.933, -0.869, 80.588, 43.045]
  MoveL 626 to (61.81, 42.94, 0) mm, rotated rx 180 ry 0 rz -39.83 deg; joints [42.868, -77.593, 86.929, -0.869, 80.589, 43.007]
  MoveL 627 to (61.08, 42.92, 0) mm, rotated rx -180 ry 0 rz -39.83 deg; joints [42.829, -77.588, 86.921, -0.869, 80.59, 42.968]
  MoveL 628 to (60.18, 42.93, 0) mm, rotated rx -180 ry 0 rz -39.83 deg; joints [42.781, -77.578, 86.908, -0.869, 80.593, 42.92]
  MoveL 629 to (59.29, 42.97, 0) mm, rotated rx 180 ry 0 rz -39.83 deg; joints [42.734, -77.566, 86.892, -0.869, 80.596, 42.872]
  MoveL 630 to (58.41, 43.02, 0) mm, rotated rx 180 ry 0 rz -39.83 deg; joints [42.687, -77.552, 86.874, -0.869, 80.6, 42.825]
  MoveL 631 to (57.52, 43.09, 0) mm, rotated rx 180 ry 0 rz -39.83 deg; joints [42.64, -77.537, 86.855, -0.869, 80.603, 42.778]
  MoveL 632 to (56.62, 43.17, 0) mm, rotated rx 180 ry 0 rz -39.83 deg; joints [42.593, -77.521, 86.834, -0.868, 80.607, 42.731]
  MoveL 633 to (55.73, 43.27, 0) mm, rotated rx 180 ry 0 rz -39.83 deg; joints [42.545, -77.503, 86.811, -0.868, 80.612, 42.683]
  MoveL 634 to (54.84, 43.41, 0) mm, rotated rx -180 ry 0 rz -39.83 deg; joints [42.499, -77.483, 86.785, -0.868, 80.617, 42.637]
  MoveL 635 to (53.96, 43.59, 0) mm, rotated rx 180 ry 0 rz -39.83 deg; joints [42.453, -77.458, 86.754, -0.868, 80.623, 42.591]
  MoveL 636 to (53.06, 43.83, 0) mm, rotated rx 180 ry 0 rz -39.83 deg; joints [42.407, -77.429, 86.716, -0.868, 80.63, 42.544]
  MoveL 637 to (52.16, 44.12, 0) mm, rotated rx -180 ry 0 rz -39.83 deg; joints [42.361, -77.396, 86.675, -0.868, 80.638, 42.499]
  MoveL 638 to (51.28, 44.43, 0) mm, rotated rx 180 ry 0 rz -39.83 deg; joints [42.316, -77.361, 86.63, -0.868, 80.646, 42.454]
  MoveL 639 to (50.39, 44.74, 0) mm, rotated rx 180 ry 0 rz -39.83 deg; joints [42.272, -77.325, 86.586, -0.868, 80.655, 42.409]
  MoveL 640 to (49.62, 45.01, 0) mm, rotated rx 180 ry 0 rz -39.83 deg; joints [42.232, -77.294, 86.547, -0.868, 80.662, 42.369]
  MoveL 641 to (48.84, 45.29, 0) mm, rotated rx 180 ry 0 rz -39.83 deg; joints [42.193, -77.263, 86.508, -0.868, 80.67, 42.33]
  MoveL 642 to (48.08, 45.58, 0) mm, rotated rx -180 ry 0 rz -39.83 deg; joints [42.155, -77.231, 86.467, -0.868, 80.678, 42.291]
  MoveL 643 to (47.33, 45.9, 0) mm, rotated rx 180 ry 0 rz -39.83 deg; joints [42.117, -77.196, 86.423, -0.868, 80.686, 42.254]
  MoveL 644 to (46.54, 46.31, 0) mm, rotated rx -180 ry 0 rz -39.83 deg; joints [42.078, -77.154, 86.371, -0.867, 80.696, 42.214]
  MoveL 645 to (45.76, 46.75, 0) mm, rotated rx 180 ry 0 rz -39.83 deg; joints [42.04, -77.109, 86.314, -0.867, 80.707, 42.177]
  MoveL 646 to (45.01, 47.23, 0) mm, rotated rx 180 ry 0 rz -39.83 deg; joints [42.004, -77.062, 86.255, -0.867, 80.718, 42.14]
  MoveL 647 to (44.26, 47.72, 0) mm, rotated rx -180 ry 0 rz -39.83 deg; joints [41.968, -77.013, 86.194, -0.867, 80.73, 42.104]
  MoveL 648 to (43.26, 48.41, 0) mm, rotated rx 180 ry 0 rz -39.83 deg; joints [41.92, -76.945, 86.109, -0.867, 80.747, 42.056]
  MoveL 649 to (42.27, 49.12, 0) mm, rotated rx -180 ry 0 rz -39.83 deg; joints [41.873, -76.876, 86.022, -0.867, 80.763, 42.008]
  MoveL 650 to (41.3, 49.85, 0) mm, rotated rx -180 ry 0 rz -39.83 deg; joints [41.828, -76.805, 85.933, -0.867, 80.781, 41.963]
  MoveL 651 to (40.37, 50.62, 0) mm, rotated rx 180 ry 0 rz -39.83 deg; joints [41.784, -76.731, 85.841, -0.867, 80.799, 41.919]
  MoveL 652 to (39.52, 51.38, 0) mm, rotated rx 180 ry 0 rz -39.83 deg; joints [41.745, -76.659, 85.75, -0.867, 80.816, 41.88]
  MoveL 653 to (38.7, 52.18, 0) mm, rotated rx 180 ry 0 rz -39.83 deg; joints [41.708, -76.585, 85.657, -0.867, 80.835, 41.842]
  MoveL 654 to (37.91, 53, 0) mm, rotated rx 180 ry 0 rz -39.83 deg; joints [41.673, -76.508, 85.561, -0.866, 80.854, 41.807]
  MoveL 655 to (37.14, 53.85, 0) mm, rotated rx 180 ry 0 rz -39.83 deg; joints [41.639, -76.43, 85.463, -0.866, 80.873, 41.773]
  MoveL 656 to (36.33, 54.79, 0) mm, rotated rx 180 ry 0 rz -39.83 deg; joints [41.604, -76.344, 85.355, -0.866, 80.895, 41.737]
  MoveL 657 to (35.54, 55.75, 0) mm, rotated rx 180 ry 0 rz -39.83 deg; joints [41.57, -76.256, 85.244, -0.866, 80.917, 41.703]
  MoveL 658 to (34.79, 56.73, 0) mm, rotated rx -180 ry 0 rz -39.83 deg; joints [41.538, -76.167, 85.132, -0.866, 80.939, 41.671]
  MoveL 659 to (34.07, 57.74, 0) mm, rotated rx 180 ry 0 rz -39.83 deg; joints [41.509, -76.076, 85.017, -0.866, 80.962, 41.641]
  MoveL 660 to (33.37, 58.81, 0) mm, rotated rx 180 ry 0 rz -39.83 deg; joints [41.481, -75.979, 84.896, -0.866, 80.987, 41.613]
  MoveL 661 to (32.72, 59.92, 0) mm, rotated rx 180 ry 0 rz -39.83 deg; joints [41.456, -75.882, 84.773, -0.866, 81.012, 41.587]
